(* Logix 5000 project; controller reports 1756-L63 rev 20.11; software revision 20.04; part 50 of 52 *)

        [182].log_data[31].max := 1.0, [182].log_data[31].total := 1629.7471, [182].log_data[31].time := 3600.0, [182].log_data[31].maxminute := 5, [182].log_data[31].valid := 1, [182].log_data[32].max := 1.0, [182].log_data[32].total := 1288.2471, [182].log_data[32].time := 3600.0, [182].log_data[32].maxminute := 2, [182].log_data[32].valid := 1, [182].log_data[33].time := 3600.0, [182].log_data[33].valid := 1, [182].log_data[34].time := 3600.0, [182].log_data[34].valid := 1, [182].log_data[35].max := 1.0, [182].log_data[35].total := 1629.7471, [182].log_data[35].time := 3600.0, [182].log_data[35].maxminute := 8, [182].log_data[35].valid := 1, [182].log_data[36].max := 1.0, [182].log_data[36].total := 1355.247, [182].log_data[36].time := 3600.0, [182].log_data[36].maxminute := 2, [182].log_data[36].valid := 1, [182].log_data[37].max := 7.52496, [182].log_data[37].total := 2850.735, [182].log_data[37].time := 3600.0, [182].log_data[37].minminute := 6, [182].log_data[37].valid := 1, [182].log_data[38].time := 3600.0, [182].log_data[38].valid := 1, [182].log_data[39].min := 0.9950596, [182].log_data[39].max := 1.0219122, [182].log_data[39].total := 3611.1082, [182].log_data[39].time := 3600.0, [182].log_data[39].minminute := 24, [182].log_data[39].maxminute := 6, [182].log_data[39].valid := 1, [182].log_data[40].min := 7.5459046, [182].log_data[40].max := 7.5849276, [182].log_data[40].total := 27253.14, [182].log_data[40].time := 3600.0, [182].log_data[40].minminute := 44, [182].log_data[40].maxminute := 47, [182].log_data[40].valid := 1, [182].log_data[41].min := 0.06945386, [182].log_data[41].max := 0.103412114, [182].log_data[41].total := 295.7068, [182].log_data[41].time := 3600.0, [182].log_data[41].minminute := 41, [182].log_data[41].valid := 1, [182].log_data[42].min := 2.292467, [182].log_data[42].max := 2.2978847, [182].log_data[42].total := 8263.784, [182].log_data[42].time := 3600.0, [182].log_data[42].minminute := 25, [182].log_data[42].valid := 1, [182].log_data[43].min := -0.26000214, [182].log_data[43].max := -0.23999786, [182].log_data[43].total := -935.9582,
        [182].log_data[43].time := 3600.0, [182].log_data[43].maxminute := 40, [182].log_data[43].valid := 1, [182].log_data[44].min := -0.30000305, [182].log_data[44].max := -0.27999878, [182].log_data[44].total := -1034.0974, [182].log_data[44].time := 3600.0, [182].log_data[44].valid := 1, [182].log_data[45].time := 3600.0, [182].log_data[45].valid := 1, [182].log_data[46].time := 3600.0, [182].log_data[46].valid := 1, [182].log_data[47].time := 3600.0, [182].log_data[47].valid := 1, [182].log_data[48].min := 6.578031, [182].log_data[48].max := 6.975128, [182].log_data[48].total := 24224.42, [182].log_data[48].time := 3600.0, [182].log_data[48].minminute := 30, [182].log_data[48].maxminute := 8, [182].log_data[48].valid := 1, [182].log_data[49].min := 6.7680936, [182].log_data[49].max := 9.480644, [182].log_data[49].total := 29086.424, [182].log_data[49].time := 3600.0, [182].log_data[49].minminute := 27, [182].log_data[49].valid := 1, [182].log_data[50].min := 2.0458467, [182].log_data[50].max := 2.1517262, [182].log_data[50].total := 7513.503, [182].log_data[50].time := 3600.0, [182].log_data[50].minminute := 58, [182].log_data[50].maxminute := 2, [182].log_data[50].valid := 1, [182].log_data[51].time := 3600.0, [182].log_data[51].valid := 1, [182].log_data[52].min := -4.199997, [182].log_data[52].max := 0.13999939, [182].log_data[52].total := -7374.407, [182].log_data[52].time := 3600.0, [182].log_data[52].minminute := 2, [182].log_data[52].maxminute := 56, [182].log_data[52].valid := 1, [182].log_data[53].min := -3.9799957, [182].log_data[53].max := 0.27999878, [182].log_data[53].total := -6905.0986, [182].log_data[53].time := 3600.0, [182].log_data[53].minminute := 2, [182].log_data[53].maxminute := 28, [182].log_data[53].valid := 1, [182].log_data[54].max := 0.538, [182].log_data[54].total := 1154.3633, [182].log_data[54].time := 3600.0, [182].log_data[54].maxminute := 16, [182].log_data[54].valid := 1, [182].log_data[55].max := 0.5285, [182].log_data[55].total := 1182.999, [182].log_data[55].time := 3600.0, [182].log_data[55].maxminute := 19, [182].log_data[55].valid := 1,
        [182].log_data[56].min := 0.16044189, [182].log_data[56].max := 0.16087373, [182].log_data[56].total := 578.1737, [182].log_data[56].time := 3600.0, [182].log_data[56].minminute := 7, [182].log_data[56].maxminute := 25, [182].log_data[56].valid := 1, [182].log_data[57].min := 0.34067667, [182].log_data[57].max := 0.34228623, [182].log_data[57].total := 1229.2501, [182].log_data[57].time := 3600.0, [182].log_data[57].minminute := 45, [182].log_data[57].maxminute := 11, [182].log_data[57].valid := 1, [182].log_data[58].time := 3600.0, [182].log_data[58].valid := 1, [182].log_data[59].time := 3600.0, [182].log_data[59].valid := 1, [182].log_data[60].valid := 1, [182].log_data[61].valid := 1, [182].log_data[62].valid := 1, [182].log_data[63].valid := 1, [182].log_data[64].valid := 1, [182].log_data[65].valid := 1, [182].log_data[66].valid := 1, [182].log_data[67].valid := 1, [182].log_data[68].valid := 1, [182].log_data[69].valid := 1, [182].log_data[70].valid := 1, [182].log_data[71].valid := 1, [182].log_data[72].valid := 1, [182].log_data[73].valid := 1, [182].log_data[74].valid := 1, [182].log_data[75].valid := 1, [182].log_data[76].valid := 1, [182].log_data[77].valid := 1, [182].log_data[78].valid := 1, [182].log_data[79].valid := 1, [182].log_data[80].valid := 1, [182].log_data[81].valid := 1, [182].log_data[82].valid := 1, [182].log_data[83].valid := 1, [182].log_data[84].valid := 1, [182].log_data[85].valid := 1, [182].log_data[86].valid := 1, [182].log_data[87].valid := 1, [182].log_data[88].valid := 1, [182].log_data[89].valid := 1, [182].log_data[90].valid := 1, [182].log_data[91].valid := 1, [182].log_data[92].valid := 1, [182].log_data[93].valid := 1, [182].log_data[94].valid := 1, [182].log_data[95].valid := 1, [182].log_data[96].valid := 1, [182].log_data[97].valid := 1, [182].log_data[98].valid := 1, [182].log_data[99].valid := 1, [182].log_data[100].valid := 1, [182].log_data[101].valid := 1,
        [182].log_data[102].valid := 1, [182].log_data[103].valid := 1, [182].log_data[104].valid := 1, [182].log_data[105].valid := 1, [182].log_data[106].valid := 1, [182].log_data[107].valid := 1, [182].log_data[108].valid := 1, [182].log_data[109].valid := 1, [182].log_data[110].valid := 1, [182].log_data[111].valid := 1, [182].log_data[112].valid := 1, [182].log_data[113].valid := 1, [182].log_data[114].valid := 1, [182].log_data[115].valid := 1, [182].log_data[116].valid := 1, [182].log_data[117].valid := 1, [182].log_data[118].valid := 1, [182].log_data[119].valid := 1, [182].log_data[120].valid := 1, [182].log_data[121].valid := 1, [182].log_data[122].valid := 1, [182].log_data[123].valid := 1, [182].log_data[124].valid := 1, [182].time.Year := 2023, [182].time.Month := 1, [182].time.Day := 12, [182].time.Hour := 9, [182].time.Minute := 59, [182].time.Second := 59, [183].log_data[0].min := 1.0, [183].log_data[0].max := 1.0, [183].log_data[0].total := 3600.0, [183].log_data[0].time := 3600.0, [183].log_data[0].valid := 1, [183].log_data[1].max := 1.0, [183].log_data[1].total := 590.5, [183].log_data[1].time := 3600.0, [183].log_data[1].maxminute := 32, [183].log_data[1].valid := 1, [183].log_data[2].max := 1.0, [183].log_data[2].total := 587.0, [183].log_data[2].time := 3600.0, [183].log_data[2].maxminute := 32, [183].log_data[2].valid := 1, [183].log_data[3].time := 3600.0, [183].log_data[3].valid := 1, [183].log_data[4].time := 3600.0, [183].log_data[4].valid := 1, [183].log_data[5].max := 1.0, [183].log_data[5].total := 226.5, [183].log_data[5].time := 3600.0, [183].log_data[5].maxminute := 34, [183].log_data[5].valid := 1, [183].log_data[6].time := 3600.0, [183].log_data[6].valid := 1, [183].log_data[7].time := 3600.0, [183].log_data[7].valid := 1, [183].log_data[8].max := 1.0, [183].log_data[8].total := 3318.0, [183].log_data[8].time := 3600.0,
        [183].log_data[8].minminute := 32, [183].log_data[8].valid := 1, [183].log_data[9].max := 1.0, [183].log_data[9].total := 3314.5, [183].log_data[9].time := 3600.0, [183].log_data[9].minminute := 32, [183].log_data[9].valid := 1, [183].log_data[10].min := 1.0, [183].log_data[10].max := 1.0, [183].log_data[10].total := 3600.0, [183].log_data[10].time := 3600.0, [183].log_data[10].valid := 1, [183].log_data[11].time := 3600.0, [183].log_data[11].valid := 1, [183].log_data[12].min := 1.0, [183].log_data[12].max := 1.0, [183].log_data[12].total := 3600.0, [183].log_data[12].time := 3600.0, [183].log_data[12].valid := 1, [183].log_data[13].min := 1.0, [183].log_data[13].max := 1.0, [183].log_data[13].total := 3600.0, [183].log_data[13].time := 3600.0, [183].log_data[13].valid := 1, [183].log_data[14].time := 3600.0, [183].log_data[14].valid := 1, [183].log_data[15].time := 3600.0, [183].log_data[15].valid := 1, [183].log_data[16].time := 3600.0, [183].log_data[16].valid := 1, [183].log_data[17].min := 1.0, [183].log_data[17].max := 1.0, [183].log_data[17].total := 3600.0, [183].log_data[17].time := 3600.0, [183].log_data[17].valid := 1, [183].log_data[18].time := 3600.0, [183].log_data[18].valid := 1, [183].log_data[19].time := 3600.0, [183].log_data[19].valid := 1, [183].log_data[20].time := 3600.0, [183].log_data[20].valid := 1, [183].log_data[21].min := 1.0, [183].log_data[21].max := 1.0, [183].log_data[21].total := 3600.0, [183].log_data[21].time := 3600.0, [183].log_data[21].valid := 1, [183].log_data[22].time := 3600.0, [183].log_data[22].valid := 1, [183].log_data[23].time := 3600.0, [183].log_data[23].valid := 1, [183].log_data[24].time := 3600.0, [183].log_data[24].valid := 1, [183].log_data[25].time := 3600.0, [183].log_data[25].valid := 1, [183].log_data[26].time := 3600.0, [183].log_data[26].valid := 1, [183].log_data[27].time := 3600.0, [183].log_data[27].valid := 1, [183].log_data[28].time := 3600.0, [183].log_data[28].valid := 1,
        [183].log_data[29].min := 1.0, [183].log_data[29].max := 1.0, [183].log_data[29].total := 3600.0, [183].log_data[29].time := 3600.0, [183].log_data[29].valid := 1, [183].log_data[30].min := 1.0, [183].log_data[30].max := 1.0, [183].log_data[30].total := 3600.0, [183].log_data[30].time := 3600.0, [183].log_data[30].valid := 1, [183].log_data[31].max := 1.0, [183].log_data[31].total := 1268.7471, [183].log_data[31].time := 3600.0, [183].log_data[31].maxminute := 8, [183].log_data[31].valid := 1, [183].log_data[32].max := 1.0, [183].log_data[32].total := 1604.7471, [183].log_data[32].time := 3600.0, [183].log_data[32].minminute := 7, [183].log_data[32].valid := 1, [183].log_data[33].time := 3600.0, [183].log_data[33].valid := 1, [183].log_data[34].time := 3600.0, [183].log_data[34].valid := 1, [183].log_data[35].max := 1.0, [183].log_data[35].total := 1172.2471, [183].log_data[35].time := 3600.0, [183].log_data[35].maxminute := 11, [183].log_data[35].valid := 1, [183].log_data[36].max := 1.0, [183].log_data[36].total := 1629.998, [183].log_data[36].time := 3600.0, [183].log_data[36].maxminute := 1, [183].log_data[36].valid := 1, [183].log_data[37].max := 6.980448, [183].log_data[37].total := 3611.7107, [183].log_data[37].time := 3600.0, [183].log_data[37].maxminute := 33, [183].log_data[37].valid := 1, [183].log_data[38].time := 3600.0, [183].log_data[38].valid := 1, [183].log_data[39].min := 0.9967084, [183].log_data[39].max := 1.0206168, [183].log_data[39].total := 3614.8816, [183].log_data[39].time := 3600.0, [183].log_data[39].minminute := 13, [183].log_data[39].maxminute := 35, [183].log_data[39].valid := 1, [183].log_data[40].min := 7.5316143, [183].log_data[40].max := 7.5849276, [183].log_data[40].total := 27245.064, [183].log_data[40].time := 3600.0, [183].log_data[40].minminute := 25, [183].log_data[40].maxminute := 52, [183].log_data[40].valid := 1, [183].log_data[41].min := 0.0686687, [183].log_data[41].max := 0.09438281, [183].log_data[41].total := 279.35208, [183].log_data[41].time := 3600.0, [183].log_data[41].minminute := 53,
        [183].log_data[41].maxminute := 2, [183].log_data[41].valid := 1, [183].log_data[42].min := 2.2927027, [183].log_data[42].max := 2.297767, [183].log_data[42].total := 8263.784, [183].log_data[42].time := 3600.0, [183].log_data[42].minminute := 5, [183].log_data[42].maxminute := 6, [183].log_data[42].valid := 1, [183].log_data[43].min := -0.26000214, [183].log_data[43].max := -0.23999786, [183].log_data[43].total := -935.8381, [183].log_data[43].time := 3600.0, [183].log_data[43].maxminute := 2, [183].log_data[43].valid := 1, [183].log_data[44].min := -0.30000305, [183].log_data[44].max := -0.27999878, [183].log_data[44].total := -1026.5973, [183].log_data[44].time := 3600.0, [183].log_data[44].valid := 1, [183].log_data[45].time := 3600.0, [183].log_data[45].valid := 1, [183].log_data[46].time := 3600.0, [183].log_data[46].valid := 1, [183].log_data[47].time := 3600.0, [183].log_data[47].valid := 1, [183].log_data[48].min := 6.5824285, [183].log_data[48].max := 6.957815, [183].log_data[48].total := 24226.725, [183].log_data[48].time := 3600.0, [183].log_data[48].minminute := 59, [183].log_data[48].maxminute := 37, [183].log_data[48].valid := 1, [183].log_data[49].min := 6.8424883, [183].log_data[49].max := 9.4459, [183].log_data[49].total := 31391.893, [183].log_data[49].time := 3600.0, [183].log_data[49].minminute := 58, [183].log_data[49].maxminute := 22, [183].log_data[49].valid := 1, [183].log_data[50].min := 1.9999144, [183].log_data[50].max := 2.1501951, [183].log_data[50].total := 7404.694, [183].log_data[50].time := 3600.0, [183].log_data[50].minminute := 32, [183].log_data[50].maxminute := 37, [183].log_data[50].valid := 1, [183].log_data[51].time := 3600.0, [183].log_data[51].valid := 1, [183].log_data[52].min := -3.8600006, [183].log_data[52].max := 0.13999939, [183].log_data[52].total := -7261.7637, [183].log_data[52].time := 3600.0, [183].log_data[52].minminute := 37, [183].log_data[52].maxminute := 7, [183].log_data[52].valid := 1, [183].log_data[53].min := -3.7200012, [183].log_data[53].max := 0.22000122, [183].log_data[53].total := -6467.2256, [183].log_data[53].time := 3600.0,
        [183].log_data[53].minminute := 37, [183].log_data[53].valid := 1, [183].log_data[54].max := 0.52349997, [183].log_data[54].total := 1138.3706, [183].log_data[54].time := 3600.0, [183].log_data[54].minminute := 7, [183].log_data[54].maxminute := 55, [183].log_data[54].valid := 1, [183].log_data[55].max := 0.5395, [183].log_data[55].total := 1109.6932, [183].log_data[55].time := 3600.0, [183].log_data[55].maxminute := 11, [183].log_data[55].valid := 1, [183].log_data[56].min := 0.16044189, [183].log_data[56].max := 0.16083448, [183].log_data[56].total := 578.1302, [183].log_data[56].time := 3600.0, [183].log_data[56].minminute := 22, [183].log_data[56].maxminute := 1, [183].log_data[56].valid := 1, [183].log_data[57].min := 0.34040186, [183].log_data[57].max := 0.34106925, [183].log_data[57].total := 1226.9022, [183].log_data[57].time := 3600.0, [183].log_data[57].minminute := 59, [183].log_data[57].maxminute := 18, [183].log_data[57].valid := 1, [183].log_data[58].time := 3600.0, [183].log_data[58].valid := 1, [183].log_data[59].time := 3600.0, [183].log_data[59].valid := 1, [183].log_data[60].valid := 1, [183].log_data[61].valid := 1, [183].log_data[62].valid := 1, [183].log_data[63].valid := 1, [183].log_data[64].valid := 1, [183].log_data[65].valid := 1, [183].log_data[66].valid := 1, [183].log_data[67].valid := 1, [183].log_data[68].valid := 1, [183].log_data[69].valid := 1, [183].log_data[70].valid := 1, [183].log_data[71].valid := 1, [183].log_data[72].valid := 1, [183].log_data[73].valid := 1, [183].log_data[74].valid := 1, [183].log_data[75].valid := 1, [183].log_data[76].valid := 1, [183].log_data[77].valid := 1, [183].log_data[78].valid := 1, [183].log_data[79].valid := 1, [183].log_data[80].valid := 1, [183].log_data[81].valid := 1, [183].log_data[82].valid := 1, [183].log_data[83].valid := 1, [183].log_data[84].valid := 1, [183].log_data[85].valid := 1, [183].log_data[86].valid := 1, [183].log_data[87].valid := 1, [183].log_data[88].valid := 1,
        [183].log_data[89].valid := 1, [183].log_data[90].valid := 1, [183].log_data[91].valid := 1, [183].log_data[92].valid := 1, [183].log_data[93].valid := 1, [183].log_data[94].valid := 1, [183].log_data[95].valid := 1, [183].log_data[96].valid := 1, [183].log_data[97].valid := 1, [183].log_data[98].valid := 1, [183].log_data[99].valid := 1, [183].log_data[100].valid := 1, [183].log_data[101].valid := 1, [183].log_data[102].valid := 1, [183].log_data[103].valid := 1, [183].log_data[104].valid := 1, [183].log_data[105].valid := 1, [183].log_data[106].valid := 1, [183].log_data[107].valid := 1, [183].log_data[108].valid := 1, [183].log_data[109].valid := 1, [183].log_data[110].valid := 1, [183].log_data[111].valid := 1, [183].log_data[112].valid := 1, [183].log_data[113].valid := 1, [183].log_data[114].valid := 1, [183].log_data[115].valid := 1, [183].log_data[116].valid := 1, [183].log_data[117].valid := 1, [183].log_data[118].valid := 1, [183].log_data[119].valid := 1, [183].log_data[120].valid := 1, [183].log_data[121].valid := 1, [183].log_data[122].valid := 1, [183].log_data[123].valid := 1, [183].log_data[124].valid := 1, [183].time.Year := 2023, [183].time.Month := 1, [183].time.Day := 12, [183].time.Hour := 10, [183].time.Minute := 59, [183].time.Second := 59, [184].log_data[0].min := 1.0, [184].log_data[0].max := 1.0, [184].log_data[0].total := 3600.0, [184].log_data[0].time := 3600.0, [184].log_data[0].valid := 1, [184].log_data[1].time := 3600.0, [184].log_data[1].valid := 1, [184].log_data[2].time := 3600.0, [184].log_data[2].valid := 1, [184].log_data[3].time := 3600.0, [184].log_data[3].valid := 1, [184].log_data[4].time := 3600.0, [184].log_data[4].valid := 1, [184].log_data[5].time := 3600.0, [184].log_data[5].valid := 1, [184].log_data[6].time := 3600.0, [184].log_data[6].valid := 1, [184].log_data[7].time := 3600.0,
        [184].log_data[7].valid := 1, [184].log_data[8].min := 1.0, [184].log_data[8].max := 1.0, [184].log_data[8].total := 3600.0, [184].log_data[8].time := 3600.0, [184].log_data[8].valid := 1, [184].log_data[9].min := 1.0, [184].log_data[9].max := 1.0, [184].log_data[9].total := 3600.0, [184].log_data[9].time := 3600.0, [184].log_data[9].valid := 1, [184].log_data[10].min := 1.0, [184].log_data[10].max := 1.0, [184].log_data[10].total := 3600.0, [184].log_data[10].time := 3600.0, [184].log_data[10].valid := 1, [184].log_data[11].time := 3600.0, [184].log_data[11].valid := 1, [184].log_data[12].min := 1.0, [184].log_data[12].max := 1.0, [184].log_data[12].total := 3600.0, [184].log_data[12].time := 3600.0, [184].log_data[12].valid := 1, [184].log_data[13].min := 1.0, [184].log_data[13].max := 1.0, [184].log_data[13].total := 3600.0, [184].log_data[13].time := 3600.0, [184].log_data[13].valid := 1, [184].log_data[14].time := 3600.0, [184].log_data[14].valid := 1, [184].log_data[15].time := 3600.0, [184].log_data[15].valid := 1, [184].log_data[16].time := 3600.0, [184].log_data[16].valid := 1, [184].log_data[17].min := 1.0, [184].log_data[17].max := 1.0, [184].log_data[17].total := 3600.0, [184].log_data[17].time := 3600.0, [184].log_data[17].valid := 1, [184].log_data[18].time := 3600.0, [184].log_data[18].valid := 1, [184].log_data[19].time := 3600.0, [184].log_data[19].valid := 1, [184].log_data[20].time := 3600.0, [184].log_data[20].valid := 1, [184].log_data[21].min := 1.0, [184].log_data[21].max := 1.0, [184].log_data[21].total := 3600.0, [184].log_data[21].time := 3600.0, [184].log_data[21].valid := 1, [184].log_data[22].time := 3600.0, [184].log_data[22].valid := 1, [184].log_data[23].time := 3600.0, [184].log_data[23].valid := 1, [184].log_data[24].time := 3600.0, [184].log_data[24].valid := 1, [184].log_data[25].time := 3600.0, [184].log_data[25].valid := 1, [184].log_data[26].time := 3600.0, [184].log_data[26].valid := 1,
        [184].log_data[27].time := 3600.0, [184].log_data[27].valid := 1, [184].log_data[28].time := 3600.0, [184].log_data[28].valid := 1, [184].log_data[29].min := 1.0, [184].log_data[29].max := 1.0, [184].log_data[29].total := 3600.0, [184].log_data[29].time := 3600.0, [184].log_data[29].valid := 1, [184].log_data[30].min := 1.0, [184].log_data[30].max := 1.0, [184].log_data[30].total := 3600.0, [184].log_data[30].time := 3600.0, [184].log_data[30].valid := 1, [184].log_data[31].max := 1.0, [184].log_data[31].total := 1629.998, [184].log_data[31].time := 3600.0, [184].log_data[31].maxminute := 5, [184].log_data[31].valid := 1, [184].log_data[32].max := 1.0, [184].log_data[32].total := 1440.498, [184].log_data[32].time := 3600.0, [184].log_data[32].minminute := 4, [184].log_data[32].valid := 1, [184].log_data[33].time := 3600.0, [184].log_data[33].valid := 1, [184].log_data[34].time := 3600.0, [184].log_data[34].valid := 1, [184].log_data[35].max := 1.0, [184].log_data[35].total := 1543.998, [184].log_data[35].time := 3600.0, [184].log_data[35].minminute := 7, [184].log_data[35].valid := 1, [184].log_data[36].max := 1.0, [184].log_data[36].total := 1614.7471, [184].log_data[36].time := 3600.0, [184].log_data[36].maxminute := 9, [184].log_data[36].valid := 1, [184].log_data[37].time := 3600.0, [184].log_data[37].valid := 1, [184].log_data[38].time := 3600.0, [184].log_data[38].valid := 1, [184].log_data[39].min := 1.000595, [184].log_data[39].max := 1.0097814, [184].log_data[39].total := 3621.283, [184].log_data[39].time := 3600.0, [184].log_data[39].minminute := 56, [184].log_data[39].maxminute := 32, [184].log_data[39].valid := 1, [184].log_data[40].min := 7.530241, [184].log_data[40].max := 7.590423, [184].log_data[40].total := 27254.365, [184].log_data[40].time := 3600.0, [184].log_data[40].minminute := 14, [184].log_data[40].maxminute := 2, [184].log_data[40].valid := 1, [184].log_data[41].min := 0.071613036, [184].log_data[41].max := 0.10674902, [184].log_data[41].total := 300.04837, [184].log_data[41].time := 3600.0,
        [184].log_data[41].minminute := 57, [184].log_data[41].maxminute := 12, [184].log_data[41].valid := 1, [184].log_data[42].min := 2.2928205, [184].log_data[42].max := 2.2978847, [184].log_data[42].total := 8263.812, [184].log_data[42].time := 3600.0, [184].log_data[42].minminute := 40, [184].log_data[42].maxminute := 35, [184].log_data[42].valid := 1, [184].log_data[43].min := -0.26000214, [184].log_data[43].max := -0.23999786, [184].log_data[43].total := -935.8931, [184].log_data[43].time := 3600.0, [184].log_data[43].maxminute := 5, [184].log_data[43].valid := 1, [184].log_data[44].min := -0.30000305, [184].log_data[44].max := -0.27999878, [184].log_data[44].total := -1037.5183, [184].log_data[44].time := 3600.0, [184].log_data[44].valid := 1, [184].log_data[45].time := 3600.0, [184].log_data[45].valid := 1, [184].log_data[46].time := 3600.0, [184].log_data[46].valid := 1, [184].log_data[47].time := 3600.0, [184].log_data[47].valid := 1, [184].log_data[48].min := 6.5766573, [184].log_data[48].max := 6.788259, [184].log_data[48].total := 24232.771, [184].log_data[48].time := 3600.0, [184].log_data[48].minminute := 2, [184].log_data[48].maxminute := 16, [184].log_data[48].valid := 1, [184].log_data[49].min := 6.8424883, [184].log_data[49].max := 9.414298, [184].log_data[49].total := 31253.555, [184].log_data[49].time := 3600.0, [184].log_data[49].maxminute := 54, [184].log_data[49].valid := 1, [184].log_data[50].min := 2.0008566, [184].log_data[50].max := 2.0907187, [184].log_data[50].total := 7364.591, [184].log_data[50].time := 3600.0, [184].log_data[50].minminute := 59, [184].log_data[50].valid := 1, [184].log_data[51].time := 3600.0, [184].log_data[51].valid := 1, [184].log_data[52].min := -2.8600006, [184].log_data[52].max := 0.13999939, [184].log_data[52].total := -7446.0986, [184].log_data[52].time := 3600.0, [184].log_data[52].minminute := 6, [184].log_data[52].maxminute := 4, [184].log_data[52].valid := 1, [184].log_data[53].min := -2.4800034, [184].log_data[53].max := 0.2599945, [184].log_data[53].total := -7103.2104, [184].log_data[53].time := 3600.0, [184].log_data[53].minminute := 21,
        [184].log_data[53].maxminute := 50, [184].log_data[53].valid := 1, [184].log_data[54].max := 0.5525, [184].log_data[54].total := 1217.0905, [184].log_data[54].time := 3600.0, [184].log_data[54].minminute := 4, [184].log_data[54].maxminute := 6, [184].log_data[54].valid := 1, [184].log_data[55].max := 0.5205, [184].log_data[55].total := 1254.2858, [184].log_data[55].time := 3600.0, [184].log_data[55].minminute := 7, [184].log_data[55].maxminute := 19, [184].log_data[55].valid := 1, [184].log_data[56].min := 0.16040264, [184].log_data[56].max := 0.16079521, [184].log_data[56].total := 578.0307, [184].log_data[56].time := 3600.0, [184].log_data[56].minminute := 26, [184].log_data[56].maxminute := 4, [184].log_data[56].valid := 1, [184].log_data[57].min := 0.33875299, [184].log_data[57].max := 0.3405589, [184].log_data[57].total := 1220.648, [184].log_data[57].time := 3600.0, [184].log_data[57].minminute := 37, [184].log_data[57].valid := 1, [184].log_data[58].time := 3600.0, [184].log_data[58].valid := 1, [184].log_data[59].time := 3600.0, [184].log_data[59].valid := 1, [184].log_data[60].valid := 1, [184].log_data[61].valid := 1, [184].log_data[62].valid := 1, [184].log_data[63].valid := 1, [184].log_data[64].valid := 1, [184].log_data[65].valid := 1, [184].log_data[66].valid := 1, [184].log_data[67].valid := 1, [184].log_data[68].valid := 1, [184].log_data[69].valid := 1, [184].log_data[70].valid := 1, [184].log_data[71].valid := 1, [184].log_data[72].valid := 1, [184].log_data[73].valid := 1, [184].log_data[74].valid := 1, [184].log_data[75].valid := 1, [184].log_data[76].valid := 1, [184].log_data[77].valid := 1, [184].log_data[78].valid := 1, [184].log_data[79].valid := 1, [184].log_data[80].valid := 1, [184].log_data[81].valid := 1, [184].log_data[82].valid := 1, [184].log_data[83].valid := 1, [184].log_data[84].valid := 1, [184].log_data[85].valid := 1, [184].log_data[86].valid := 1, [184].log_data[87].valid := 1, [184].log_data[88].valid := 1,
        [184].log_data[89].valid := 1, [184].log_data[90].valid := 1, [184].log_data[91].valid := 1, [184].log_data[92].valid := 1, [184].log_data[93].valid := 1, [184].log_data[94].valid := 1, [184].log_data[95].valid := 1, [184].log_data[96].valid := 1, [184].log_data[97].valid := 1, [184].log_data[98].valid := 1, [184].log_data[99].valid := 1, [184].log_data[100].valid := 1, [184].log_data[101].valid := 1, [184].log_data[102].valid := 1, [184].log_data[103].valid := 1, [184].log_data[104].valid := 1, [184].log_data[105].valid := 1, [184].log_data[106].valid := 1, [184].log_data[107].valid := 1, [184].log_data[108].valid := 1, [184].log_data[109].valid := 1, [184].log_data[110].valid := 1, [184].log_data[111].valid := 1, [184].log_data[112].valid := 1, [184].log_data[113].valid := 1, [184].log_data[114].valid := 1, [184].log_data[115].valid := 1, [184].log_data[116].valid := 1, [184].log_data[117].valid := 1, [184].log_data[118].valid := 1, [184].log_data[119].valid := 1, [184].log_data[120].valid := 1, [184].log_data[121].valid := 1, [184].log_data[122].valid := 1, [184].log_data[123].valid := 1, [184].log_data[124].valid := 1, [184].time.Year := 2023, [184].time.Month := 1, [184].time.Day := 12, [184].time.Hour := 11, [184].time.Minute := 59, [184].time.Second := 59, [185].log_data[0].min := 1.0, [185].log_data[0].max := 1.0, [185].log_data[0].total := 3600.0, [185].log_data[0].time := 3600.0, [185].log_data[0].valid := 1, [185].log_data[1].max := 1.0, [185].log_data[1].total := 552.5, [185].log_data[1].time := 3600.0, [185].log_data[1].maxminute := 5, [185].log_data[1].valid := 1, [185].log_data[2].max := 1.0, [185].log_data[2].total := 549.0, [185].log_data[2].time := 3600.0, [185].log_data[2].maxminute := 5, [185].log_data[2].valid := 1, [185].log_data[3].time := 3600.0, [185].log_data[3].valid := 1, [185].log_data[4].time := 3600.0,
        [185].log_data[4].valid := 1, [185].log_data[5].max := 1.0, [185].log_data[5].total := 252.0, [185].log_data[5].time := 3600.0, [185].log_data[5].maxminute := 7, [185].log_data[5].valid := 1, [185].log_data[6].time := 3600.0, [185].log_data[6].valid := 1, [185].log_data[7].time := 3600.0, [185].log_data[7].valid := 1, [185].log_data[8].max := 1.0, [185].log_data[8].total := 3070.5, [185].log_data[8].time := 3600.0, [185].log_data[8].valid := 1, [185].log_data[9].max := 1.0, [185].log_data[9].total := 3067.0, [185].log_data[9].time := 3600.0, [185].log_data[9].valid := 1, [185].log_data[10].min := 1.0, [185].log_data[10].max := 1.0, [185].log_data[10].total := 3600.0, [185].log_data[10].time := 3600.0, [185].log_data[10].valid := 1, [185].log_data[11].time := 3600.0, [185].log_data[11].valid := 1, [185].log_data[12].min := 1.0, [185].log_data[12].max := 1.0, [185].log_data[12].total := 3600.0, [185].log_data[12].time := 3600.0, [185].log_data[12].valid := 1, [185].log_data[13].min := 1.0, [185].log_data[13].max := 1.0, [185].log_data[13].total := 3600.0, [185].log_data[13].time := 3600.0, [185].log_data[13].valid := 1, [185].log_data[14].time := 3600.0, [185].log_data[14].valid := 1, [185].log_data[15].time := 3600.0, [185].log_data[15].valid := 1, [185].log_data[16].time := 3600.0, [185].log_data[16].valid := 1, [185].log_data[17].min := 1.0, [185].log_data[17].max := 1.0, [185].log_data[17].total := 3600.0, [185].log_data[17].time := 3600.0, [185].log_data[17].valid := 1, [185].log_data[18].time := 3600.0, [185].log_data[18].valid := 1, [185].log_data[19].time := 3600.0, [185].log_data[19].valid := 1, [185].log_data[20].time := 3600.0, [185].log_data[20].valid := 1, [185].log_data[21].min := 1.0, [185].log_data[21].max := 1.0, [185].log_data[21].total := 3600.0, [185].log_data[21].time := 3600.0, [185].log_data[21].valid := 1, [185].log_data[22].time := 3600.0, [185].log_data[22].valid := 1, [185].log_data[23].time := 3600.0,
        [185].log_data[23].valid := 1, [185].log_data[24].time := 3600.0, [185].log_data[24].valid := 1, [185].log_data[25].time := 3600.0, [185].log_data[25].valid := 1, [185].log_data[26].time := 3600.0, [185].log_data[26].valid := 1, [185].log_data[27].time := 3600.0, [185].log_data[27].valid := 1, [185].log_data[28].time := 3600.0, [185].log_data[28].valid := 1, [185].log_data[29].min := 1.0, [185].log_data[29].max := 1.0, [185].log_data[29].total := 3600.0, [185].log_data[29].time := 3600.0, [185].log_data[29].valid := 1, [185].log_data[30].min := 1.0, [185].log_data[30].max := 1.0, [185].log_data[30].total := 3600.0, [185].log_data[30].time := 3600.0, [185].log_data[30].valid := 1, [185].log_data[31].max := 1.0, [185].log_data[31].total := 1522.247, [185].log_data[31].time := 3600.0, [185].log_data[31].maxminute := 9, [185].log_data[31].valid := 1, [185].log_data[32].max := 1.0, [185].log_data[32].total := 1112.0, [185].log_data[32].time := 3600.0, [185].log_data[32].valid := 1, [185].log_data[33].time := 3600.0, [185].log_data[33].valid := 1, [185].log_data[34].time := 3600.0, [185].log_data[34].valid := 1, [185].log_data[35].max := 1.0, [185].log_data[35].total := 1598.498, [185].log_data[35].time := 3600.0, [185].log_data[35].maxminute := 9, [185].log_data[35].valid := 1, [185].log_data[36].max := 1.0, [185].log_data[36].total := 1102.0, [185].log_data[36].time := 3600.0, [185].log_data[36].valid := 1, [185].log_data[37].max := 7.5520477, [185].log_data[37].total := 3618.2432, [185].log_data[37].time := 3600.0, [185].log_data[37].maxminute := 6, [185].log_data[37].valid := 1, [185].log_data[38].time := 3600.0, [185].log_data[38].valid := 1, [185].log_data[39].min := 0.99694395, [185].log_data[39].max := 1.0217944, [185].log_data[39].total := 3616.0115, [185].log_data[39].time := 3600.0, [185].log_data[39].minminute := 58, [185].log_data[39].maxminute := 11, [185].log_data[39].valid := 1, [185].log_data[40].min := 7.5373855, [185].log_data[40].max := 7.590698, [185].log_data[40].total := 27249.404,
        [185].log_data[40].time := 3600.0, [185].log_data[40].minminute := 26, [185].log_data[40].maxminute := 12, [185].log_data[40].valid := 1, [185].log_data[41].min := 0.058461428, [185].log_data[41].max := 0.09948633, [185].log_data[41].total := 278.58185, [185].log_data[41].time := 3600.0, [185].log_data[41].minminute := 55, [185].log_data[41].maxminute := 19, [185].log_data[41].valid := 1, [185].log_data[42].min := 2.2929382, [185].log_data[42].max := 2.297767, [185].log_data[42].total := 8263.846, [185].log_data[42].time := 3600.0, [185].log_data[42].minminute := 51, [185].log_data[42].maxminute := 19, [185].log_data[42].valid := 1, [185].log_data[43].min := -0.26000214, [185].log_data[43].max := -0.23999786, [185].log_data[43].total := -935.95825, [185].log_data[43].time := 3600.0, [185].log_data[43].maxminute := 18, [185].log_data[43].valid := 1, [185].log_data[44].min := -0.30000305, [185].log_data[44].max := -0.27999878, [185].log_data[44].total := -1048.6907, [185].log_data[44].time := 3600.0, [185].log_data[44].valid := 1, [185].log_data[45].time := 3600.0, [185].log_data[45].valid := 1, [185].log_data[46].time := 3600.0, [185].log_data[46].valid := 1, [185].log_data[47].time := 3600.0, [185].log_data[47].valid := 1, [185].log_data[48].min := 6.5722604, [185].log_data[48].max := 6.9732046, [185].log_data[48].total := 24212.016, [185].log_data[48].time := 3600.0, [185].log_data[48].minminute := 36, [185].log_data[48].maxminute := 14, [185].log_data[48].valid := 1, [185].log_data[49].min := 6.660133, [185].log_data[49].max := 9.409195, [185].log_data[49].total := 28331.281, [185].log_data[49].time := 3600.0, [185].log_data[49].minminute := 35, [185].log_data[49].maxminute := 6, [185].log_data[49].valid := 1, [185].log_data[50].min := 1.9985011, [185].log_data[50].max := 2.1512551, [185].log_data[50].total := 7526.405, [185].log_data[50].time := 3600.0, [185].log_data[50].maxminute := 9, [185].log_data[50].valid := 1, [185].log_data[51].time := 3600.0, [185].log_data[51].valid := 1, [185].log_data[52].min := -4.040001, [185].log_data[52].max := 0.11999512, [185].log_data[52].total := -7068.036,
        [185].log_data[52].time := 3600.0, [185].log_data[52].minminute := 9, [185].log_data[52].maxminute := 16, [185].log_data[52].valid := 1, [185].log_data[53].min := -3.9799957, [185].log_data[53].max := 0.22000122, [185].log_data[53].total := -6659.7754, [185].log_data[53].time := 3600.0, [185].log_data[53].minminute := 9, [185].log_data[53].maxminute := 19, [185].log_data[53].valid := 1, [185].log_data[54].max := 0.531, [185].log_data[54].total := 1045.1531, [185].log_data[54].time := 3600.0, [185].log_data[54].maxminute := 28, [185].log_data[54].valid := 1, [185].log_data[55].max := 0.559, [185].log_data[55].total := 1071.3711, [185].log_data[55].time := 3600.0, [185].log_data[55].maxminute := 51, [185].log_data[55].valid := 1, [185].log_data[56].min := 0.16036338, [185].log_data[56].max := 0.16075596, [185].log_data[56].total := 577.9964, [185].log_data[56].time := 3600.0, [185].log_data[56].minminute := 38, [185].log_data[56].valid := 1, [185].log_data[57].min := 0.33655453, [185].log_data[57].max := 0.33918485, [185].log_data[57].total := 1217.2412, [185].log_data[57].time := 3600.0, [185].log_data[57].minminute := 51, [185].log_data[57].maxminute := 21, [185].log_data[57].valid := 1, [185].log_data[58].time := 3600.0, [185].log_data[58].valid := 1, [185].log_data[59].time := 3600.0, [185].log_data[59].valid := 1, [185].log_data[60].valid := 1, [185].log_data[61].valid := 1, [185].log_data[62].valid := 1, [185].log_data[63].valid := 1, [185].log_data[64].valid := 1, [185].log_data[65].valid := 1, [185].log_data[66].valid := 1, [185].log_data[67].valid := 1, [185].log_data[68].valid := 1, [185].log_data[69].valid := 1, [185].log_data[70].valid := 1, [185].log_data[71].valid := 1, [185].log_data[72].valid := 1, [185].log_data[73].valid := 1, [185].log_data[74].valid := 1, [185].log_data[75].valid := 1, [185].log_data[76].valid := 1, [185].log_data[77].valid := 1, [185].log_data[78].valid := 1, [185].log_data[79].valid := 1, [185].log_data[80].valid := 1, [185].log_data[81].valid := 1,
        [185].log_data[82].valid := 1, [185].log_data[83].valid := 1, [185].log_data[84].valid := 1, [185].log_data[85].valid := 1, [185].log_data[86].valid := 1, [185].log_data[87].valid := 1, [185].log_data[88].valid := 1, [185].log_data[89].valid := 1, [185].log_data[90].valid := 1, [185].log_data[91].valid := 1, [185].log_data[92].valid := 1, [185].log_data[93].valid := 1, [185].log_data[94].valid := 1, [185].log_data[95].valid := 1, [185].log_data[96].valid := 1, [185].log_data[97].valid := 1, [185].log_data[98].valid := 1, [185].log_data[99].valid := 1, [185].log_data[100].valid := 1, [185].log_data[101].valid := 1, [185].log_data[102].valid := 1, [185].log_data[103].valid := 1, [185].log_data[104].valid := 1, [185].log_data[105].valid := 1, [185].log_data[106].valid := 1, [185].log_data[107].valid := 1, [185].log_data[108].valid := 1, [185].log_data[109].valid := 1, [185].log_data[110].valid := 1, [185].log_data[111].valid := 1, [185].log_data[112].valid := 1, [185].log_data[113].valid := 1, [185].log_data[114].valid := 1, [185].log_data[115].valid := 1, [185].log_data[116].valid := 1, [185].log_data[117].valid := 1, [185].log_data[118].valid := 1, [185].log_data[119].valid := 1, [185].log_data[120].valid := 1, [185].log_data[121].valid := 1, [185].log_data[122].valid := 1, [185].log_data[123].valid := 1, [185].log_data[124].valid := 1, [185].time.Year := 2023, [185].time.Month := 1, [185].time.Day := 12, [185].time.Hour := 12, [185].time.Minute := 59, [185].time.Second := 59, [186].log_data[0].min := 1.0, [186].log_data[0].max := 1.0, [186].log_data[0].total := 3599.5, [186].log_data[0].time := 3599.5, [186].log_data[0].valid := 1, [186].log_data[1].max := 1.0, [186].log_data[1].total := 344.749, [186].log_data[1].time := 3599.5, [186].log_data[1].maxminute := 54, [186].log_data[1].valid := 1, [186].log_data[2].max := 1.0,
        [186].log_data[2].total := 341.249, [186].log_data[2].time := 3599.5, [186].log_data[2].maxminute := 54, [186].log_data[2].valid := 1, [186].log_data[3].time := 3599.5, [186].log_data[3].valid := 1, [186].log_data[4].time := 3599.5, [186].log_data[4].valid := 1, [186].log_data[5].max := 1.0, [186].log_data[5].total := 122.5, [186].log_data[5].time := 3599.5, [186].log_data[5].maxminute := 56, [186].log_data[5].valid := 1, [186].log_data[6].time := 3599.5, [186].log_data[6].valid := 1, [186].log_data[7].time := 3599.5, [186].log_data[7].valid := 1, [186].log_data[8].max := 1.0, [186].log_data[8].total := 2593.0, [186].log_data[8].time := 3599.5, [186].log_data[8].minminute := 41, [186].log_data[8].valid := 1, [186].log_data[9].max := 1.0, [186].log_data[9].total := 2589.5, [186].log_data[9].time := 3599.5, [186].log_data[9].minminute := 41, [186].log_data[9].valid := 1, [186].log_data[10].min := 1.0, [186].log_data[10].max := 1.0, [186].log_data[10].total := 3599.5, [186].log_data[10].time := 3599.5, [186].log_data[10].valid := 1, [186].log_data[11].time := 3599.5, [186].log_data[11].valid := 1, [186].log_data[12].min := 1.0, [186].log_data[12].max := 1.0, [186].log_data[12].total := 3599.5, [186].log_data[12].time := 3599.5, [186].log_data[12].valid := 1, [186].log_data[13].min := 1.0, [186].log_data[13].max := 1.0, [186].log_data[13].total := 3599.5, [186].log_data[13].time := 3599.5, [186].log_data[13].valid := 1, [186].log_data[14].time := 3599.5, [186].log_data[14].valid := 1, [186].log_data[15].time := 3599.5, [186].log_data[15].valid := 1, [186].log_data[16].time := 3599.5, [186].log_data[16].valid := 1, [186].log_data[17].min := 1.0, [186].log_data[17].max := 1.0, [186].log_data[17].total := 3599.5, [186].log_data[17].time := 3599.5, [186].log_data[17].valid := 1, [186].log_data[18].time := 3599.5, [186].log_data[18].valid := 1, [186].log_data[19].time := 3599.5, [186].log_data[19].valid := 1, [186].log_data[20].time := 3599.5,
        [186].log_data[20].valid := 1, [186].log_data[21].min := 1.0, [186].log_data[21].max := 1.0, [186].log_data[21].total := 3599.5, [186].log_data[21].time := 3599.5, [186].log_data[21].valid := 1, [186].log_data[22].time := 3599.5, [186].log_data[22].valid := 1, [186].log_data[23].time := 3599.5, [186].log_data[23].valid := 1, [186].log_data[24].time := 3599.5, [186].log_data[24].valid := 1, [186].log_data[25].time := 3599.5, [186].log_data[25].valid := 1, [186].log_data[26].time := 3599.5, [186].log_data[26].valid := 1, [186].log_data[27].time := 3599.5, [186].log_data[27].valid := 1, [186].log_data[28].time := 3599.5, [186].log_data[28].valid := 1, [186].log_data[29].min := 1.0, [186].log_data[29].max := 1.0, [186].log_data[29].total := 3599.5, [186].log_data[29].time := 3599.5, [186].log_data[29].valid := 1, [186].log_data[30].min := 1.0, [186].log_data[30].max := 1.0, [186].log_data[30].total := 3599.5, [186].log_data[30].time := 3599.5, [186].log_data[30].valid := 1, [186].log_data[31].max := 1.0, [186].log_data[31].total := 1086.498, [186].log_data[31].time := 3599.5, [186].log_data[31].maxminute := 10, [186].log_data[31].valid := 1, [186].log_data[32].max := 1.0, [186].log_data[32].total := 1186.2471, [186].log_data[32].time := 3599.5, [186].log_data[32].valid := 1, [186].log_data[33].time := 3599.5, [186].log_data[33].valid := 1, [186].log_data[34].time := 3599.5, [186].log_data[34].valid := 1, [186].log_data[35].max := 1.0, [186].log_data[35].total := 1050.498, [186].log_data[35].time := 3599.5, [186].log_data[35].valid := 1, [186].log_data[36].max := 1.0, [186].log_data[36].total := 1153.7471, [186].log_data[36].time := 3599.5, [186].log_data[36].maxminute := 2, [186].log_data[36].valid := 1, [186].log_data[37].max := 6.989477, [186].log_data[37].total := 2357.3582, [186].log_data[37].time := 3599.5, [186].log_data[37].maxminute := 55, [186].log_data[37].valid := 1, [186].log_data[38].time := 3599.5, [186].log_data[38].valid := 1, [186].log_data[39].min := 0.99753284,
        [186].log_data[39].max := 1.0212055, [186].log_data[39].total := 3613.32, [186].log_data[39].time := 3599.5, [186].log_data[39].minminute := 36, [186].log_data[39].maxminute := 56, [186].log_data[39].valid := 1, [186].log_data[40].min := 7.5459046, [186].log_data[40].max := 7.5934467, [186].log_data[40].total := 27253.635, [186].log_data[40].time := 3599.5, [186].log_data[40].maxminute := 5, [186].log_data[40].valid := 1, [186].log_data[41].min := 0.056498535, [186].log_data[41].max := 0.08829786, [186].log_data[41].total := 249.71246, [186].log_data[41].time := 3599.5, [186].log_data[41].minminute := 20, [186].log_data[41].maxminute := 23, [186].log_data[41].valid := 1, [186].log_data[42].min := 2.292467, [186].log_data[42].max := 2.297767, [186].log_data[42].total := 8262.826, [186].log_data[42].time := 3599.5, [186].log_data[42].minminute := 39, [186].log_data[42].maxminute := 44, [186].log_data[42].valid := 1, [186].log_data[43].min := -0.26000214, [186].log_data[43].max := -0.26000214, [186].log_data[43].total := -935.8432, [186].log_data[43].time := 3599.5, [186].log_data[43].valid := 1, [186].log_data[44].min := -0.30000305, [186].log_data[44].max := -0.27999878, [186].log_data[44].total := -1052.3257, [186].log_data[44].time := 3599.5, [186].log_data[44].valid := 1, [186].log_data[45].time := 3599.5, [186].log_data[45].valid := 1, [186].log_data[46].time := 3599.5, [186].log_data[46].valid := 1, [186].log_data[47].time := 3599.5, [186].log_data[47].valid := 1, [186].log_data[48].min := 6.743465, [186].log_data[48].max := 6.903678, [186].log_data[48].total := 24325.06, [186].log_data[48].time := 3599.5, [186].log_data[48].minminute := 44, [186].log_data[48].maxminute := 59, [186].log_data[48].valid := 1, [186].log_data[49].min := 8.798139, [186].log_data[49].max := 9.401342, [186].log_data[49].total := 33422.215, [186].log_data[49].time := 3599.5, [186].log_data[49].minminute := 59, [186].log_data[49].maxminute := 32, [186].log_data[49].valid := 1, [186].log_data[50].min := 1.9987367, [186].log_data[50].max := 2.1501951, [186].log_data[50].total := 7385.422, [186].log_data[50].time := 3599.5,
        [186].log_data[50].minminute := 41, [186].log_data[50].maxminute := 58, [186].log_data[50].valid := 1, [186].log_data[51].time := 3599.5, [186].log_data[51].valid := 1, [186].log_data[52].min := -4.119995, [186].log_data[52].max := 0.13999939, [186].log_data[52].total := -6856.9106, [186].log_data[52].time := 3599.5, [186].log_data[52].minminute := 58, [186].log_data[52].maxminute := 9, [186].log_data[52].valid := 1, [186].log_data[53].min := -3.899994, [186].log_data[53].max := 0.22000122, [186].log_data[53].total := -6188.398, [186].log_data[53].time := 3599.5, [186].log_data[53].minminute := 58, [186].log_data[53].maxminute := 2, [186].log_data[53].valid := 1, [186].log_data[54].max := 0.518, [186].log_data[54].total := 899.5263, [186].log_data[54].time := 3599.5, [186].log_data[54].maxminute := 10, [186].log_data[54].valid := 1, [186].log_data[55].max := 0.5335, [186].log_data[55].total := 872.8351, [186].log_data[55].time := 3599.5, [186].log_data[55].maxminute := 12, [186].log_data[55].valid := 1, [186].log_data[56].min := 0.16040264, [186].log_data[56].max := 0.16079521, [186].log_data[56].total := 577.93945, [186].log_data[56].time := 3599.5, [186].log_data[56].minminute := 47, [186].log_data[56].maxminute := 5, [186].log_data[56].valid := 1, [186].log_data[57].min := 0.33655453, [186].log_data[57].max := 0.3369471, [186].log_data[57].total := 1211.9497, [186].log_data[57].time := 3599.5, [186].log_data[57].minminute := 2, [186].log_data[57].maxminute := 9, [186].log_data[57].valid := 1, [186].log_data[58].time := 3599.5, [186].log_data[58].valid := 1, [186].log_data[59].time := 3599.5, [186].log_data[59].valid := 1, [186].log_data[60].valid := 1, [186].log_data[61].valid := 1, [186].log_data[62].valid := 1, [186].log_data[63].valid := 1, [186].log_data[64].valid := 1, [186].log_data[65].valid := 1, [186].log_data[66].valid := 1, [186].log_data[67].valid := 1, [186].log_data[68].valid := 1, [186].log_data[69].valid := 1, [186].log_data[70].valid := 1, [186].log_data[71].valid := 1, [186].log_data[72].valid := 1,
        [186].log_data[73].valid := 1, [186].log_data[74].valid := 1, [186].log_data[75].valid := 1, [186].log_data[76].valid := 1, [186].log_data[77].valid := 1, [186].log_data[78].valid := 1, [186].log_data[79].valid := 1, [186].log_data[80].valid := 1, [186].log_data[81].valid := 1, [186].log_data[82].valid := 1, [186].log_data[83].valid := 1, [186].log_data[84].valid := 1, [186].log_data[85].valid := 1, [186].log_data[86].valid := 1, [186].log_data[87].valid := 1, [186].log_data[88].valid := 1, [186].log_data[89].valid := 1, [186].log_data[90].valid := 1, [186].log_data[91].valid := 1, [186].log_data[92].valid := 1, [186].log_data[93].valid := 1, [186].log_data[94].valid := 1, [186].log_data[95].valid := 1, [186].log_data[96].valid := 1, [186].log_data[97].valid := 1, [186].log_data[98].valid := 1, [186].log_data[99].valid := 1, [186].log_data[100].valid := 1, [186].log_data[101].valid := 1, [186].log_data[102].valid := 1, [186].log_data[103].valid := 1, [186].log_data[104].valid := 1, [186].log_data[105].valid := 1, [186].log_data[106].valid := 1, [186].log_data[107].valid := 1, [186].log_data[108].valid := 1, [186].log_data[109].valid := 1, [186].log_data[110].valid := 1, [186].log_data[111].valid := 1, [186].log_data[112].valid := 1, [186].log_data[113].valid := 1, [186].log_data[114].valid := 1, [186].log_data[115].valid := 1, [186].log_data[116].valid := 1, [186].log_data[117].valid := 1, [186].log_data[118].valid := 1, [186].log_data[119].valid := 1, [186].log_data[120].valid := 1, [186].log_data[121].valid := 1, [186].log_data[122].valid := 1, [186].log_data[123].valid := 1, [186].log_data[124].valid := 1, [186].time.Year := 2023, [186].time.Month := 1, [186].time.Day := 12, [186].time.Hour := 13, [186].time.Minute := 59, [186].time.Second := 59, [187].log_data[0].min := 1.0, [187].log_data[0].max := 1.0,
        [187].log_data[0].total := 3600.0, [187].log_data[0].time := 3600.0, [187].log_data[0].valid := 1, [187].log_data[1].max := 1.0, [187].log_data[1].total := 228.251, [187].log_data[1].time := 3600.0, [187].log_data[1].minminute := 3, [187].log_data[1].valid := 1, [187].log_data[2].max := 1.0, [187].log_data[2].total := 228.251, [187].log_data[2].time := 3600.0, [187].log_data[2].minminute := 3, [187].log_data[2].valid := 1, [187].log_data[3].time := 3600.0, [187].log_data[3].valid := 1, [187].log_data[4].time := 3600.0, [187].log_data[4].valid := 1, [187].log_data[5].max := 1.0, [187].log_data[5].total := 110.0, [187].log_data[5].time := 3600.0, [187].log_data[5].maxminute := 1, [187].log_data[5].valid := 1, [187].log_data[6].time := 3600.0, [187].log_data[6].valid := 1, [187].log_data[7].time := 3600.0, [187].log_data[7].valid := 1, [187].log_data[8].min := 1.0, [187].log_data[8].max := 1.0, [187].log_data[8].total := 3600.0, [187].log_data[8].time := 3600.0, [187].log_data[8].valid := 1, [187].log_data[9].min := 1.0, [187].log_data[9].max := 1.0, [187].log_data[9].total := 3600.0, [187].log_data[9].time := 3600.0, [187].log_data[9].valid := 1, [187].log_data[10].min := 1.0, [187].log_data[10].max := 1.0, [187].log_data[10].total := 3600.0, [187].log_data[10].time := 3600.0, [187].log_data[10].valid := 1, [187].log_data[11].time := 3600.0, [187].log_data[11].valid := 1, [187].log_data[12].min := 1.0, [187].log_data[12].max := 1.0, [187].log_data[12].total := 3600.0, [187].log_data[12].time := 3600.0, [187].log_data[12].valid := 1, [187].log_data[13].min := 1.0, [187].log_data[13].max := 1.0, [187].log_data[13].total := 3600.0, [187].log_data[13].time := 3600.0, [187].log_data[13].valid := 1, [187].log_data[14].time := 3600.0, [187].log_data[14].valid := 1, [187].log_data[15].time := 3600.0, [187].log_data[15].valid := 1, [187].log_data[16].time := 3600.0, [187].log_data[16].valid := 1, [187].log_data[17].min := 1.0,
        [187].log_data[17].max := 1.0, [187].log_data[17].total := 3600.0, [187].log_data[17].time := 3600.0, [187].log_data[17].valid := 1, [187].log_data[18].time := 3600.0, [187].log_data[18].valid := 1, [187].log_data[19].time := 3600.0, [187].log_data[19].valid := 1, [187].log_data[20].time := 3600.0, [187].log_data[20].valid := 1, [187].log_data[21].min := 1.0, [187].log_data[21].max := 1.0, [187].log_data[21].total := 3600.0, [187].log_data[21].time := 3600.0, [187].log_data[21].valid := 1, [187].log_data[22].time := 3600.0, [187].log_data[22].valid := 1, [187].log_data[23].time := 3600.0, [187].log_data[23].valid := 1, [187].log_data[24].time := 3600.0, [187].log_data[24].valid := 1, [187].log_data[25].time := 3600.0, [187].log_data[25].valid := 1, [187].log_data[26].time := 3600.0, [187].log_data[26].valid := 1, [187].log_data[27].time := 3600.0, [187].log_data[27].valid := 1, [187].log_data[28].time := 3600.0, [187].log_data[28].valid := 1, [187].log_data[29].min := 1.0, [187].log_data[29].max := 1.0, [187].log_data[29].total := 3600.0, [187].log_data[29].time := 3600.0, [187].log_data[29].valid := 1, [187].log_data[30].min := 1.0, [187].log_data[30].max := 1.0, [187].log_data[30].total := 3600.0, [187].log_data[30].time := 3600.0, [187].log_data[30].valid := 1, [187].log_data[31].max := 1.0, [187].log_data[31].total := 1628.7471, [187].log_data[31].time := 3600.0, [187].log_data[31].maxminute := 8, [187].log_data[31].valid := 1, [187].log_data[32].max := 1.0, [187].log_data[32].total := 1530.249, [187].log_data[32].time := 3600.0, [187].log_data[32].minminute := 7, [187].log_data[32].valid := 1, [187].log_data[33].time := 3600.0, [187].log_data[33].valid := 1, [187].log_data[34].time := 3600.0, [187].log_data[34].valid := 1, [187].log_data[35].max := 1.0, [187].log_data[35].total := 1629.7471, [187].log_data[35].time := 3600.0, [187].log_data[35].valid := 1, [187].log_data[36].max := 1.0, [187].log_data[36].total := 1469.7471, [187].log_data[36].time := 3600.0,
        [187].log_data[36].maxminute := 11, [187].log_data[36].valid := 1, [187].log_data[37].max := 6.8296957, [187].log_data[37].total := 1124.0454, [187].log_data[37].time := 3600.0, [187].log_data[37].minminute := 2, [187].log_data[37].valid := 1, [187].log_data[38].time := 3600.0, [187].log_data[38].valid := 1, [187].log_data[39].min := 0.9972973, [187].log_data[39].max := 1.0217944, [187].log_data[39].total := 3614.423, [187].log_data[39].time := 3600.0, [187].log_data[39].minminute := 56, [187].log_data[39].maxminute := 1, [187].log_data[39].valid := 1, [187].log_data[40].min := 7.560194, [187].log_data[40].max := 7.5791564, [187].log_data[40].total := 27260.762, [187].log_data[40].time := 3600.0, [187].log_data[40].minminute := 47, [187].log_data[40].maxminute := 52, [187].log_data[40].valid := 1, [187].log_data[41].min := 0.06258349, [187].log_data[41].max := 0.09850488, [187].log_data[41].total := 288.1612, [187].log_data[41].time := 3600.0, [187].log_data[41].minminute := 54, [187].log_data[41].maxminute := 6, [187].log_data[41].valid := 1, [187].log_data[42].min := 2.2929382, [187].log_data[42].max := 2.2976491, [187].log_data[42].total := 8264.025, [187].log_data[42].time := 3600.0, [187].log_data[42].minminute := 14, [187].log_data[42].maxminute := 8, [187].log_data[42].valid := 1, [187].log_data[43].min := -0.26000214, [187].log_data[43].max := -0.23999786, [187].log_data[43].total := -935.93317, [187].log_data[43].time := 3600.0, [187].log_data[43].maxminute := 8, [187].log_data[43].valid := 1, [187].log_data[44].min := -0.30000305, [187].log_data[44].max := -0.27999878, [187].log_data[44].total := -1031.8707, [187].log_data[44].time := 3600.0, [187].log_data[44].valid := 1, [187].log_data[45].time := 3600.0, [187].log_data[45].valid := 1, [187].log_data[46].time := 3600.0, [187].log_data[46].valid := 1, [187].log_data[47].time := 3600.0, [187].log_data[47].valid := 1, [187].log_data[48].min := 6.5777564, [187].log_data[48].max := 6.946274, [187].log_data[48].total := 24229.58, [187].log_data[48].time := 3600.0, [187].log_data[48].minminute := 25, [187].log_data[48].maxminute := 3,
        [187].log_data[48].valid := 1, [187].log_data[49].min := 6.675248, [187].log_data[49].max := 9.249413, [187].log_data[49].total := 28529.777, [187].log_data[49].time := 3600.0, [187].log_data[49].minminute := 22, [187].log_data[49].maxminute := 59, [187].log_data[49].valid := 1, [187].log_data[50].min := 2.0300648, [187].log_data[50].max := 2.1118004, [187].log_data[50].total := 7468.97, [187].log_data[50].time := 3600.0, [187].log_data[50].minminute := 59, [187].log_data[50].maxminute := 5, [187].log_data[50].valid := 1, [187].log_data[51].time := 3600.0, [187].log_data[51].valid := 1, [187].log_data[52].min := -2.9199982, [187].log_data[52].max := 0.13999939, [187].log_data[52].total := -7671.008, [187].log_data[52].time := 3600.0, [187].log_data[52].minminute := 8, [187].log_data[52].maxminute := 7, [187].log_data[52].valid := 1, [187].log_data[53].min := -2.4800034, [187].log_data[53].max := 0.22000122, [187].log_data[53].total := -6891.756, [187].log_data[53].time := 3600.0, [187].log_data[53].minminute := 1, [187].log_data[53].maxminute := 10, [187].log_data[53].valid := 1, [187].log_data[54].max := 0.546, [187].log_data[54].total := 1254.6321, [187].log_data[54].time := 3600.0, [187].log_data[54].minminute := 7, [187].log_data[54].maxminute := 8, [187].log_data[54].valid := 1, [187].log_data[55].max := 0.54249996, [187].log_data[55].total := 1228.7072, [187].log_data[55].time := 3600.0, [187].log_data[55].maxminute := 22, [187].log_data[55].valid := 1, [187].log_data[56].min := 0.16036338, [187].log_data[56].max := 0.16079521, [187].log_data[56].total := 577.9204, [187].log_data[56].time := 3600.0, [187].log_data[56].minminute := 15, [187].log_data[56].maxminute := 7, [187].log_data[56].valid := 1, [187].log_data[57].min := 0.33474863, [187].log_data[57].max := 0.3369471, [187].log_data[57].total := 1208.6879, [187].log_data[57].time := 3600.0, [187].log_data[57].minminute := 49, [187].log_data[57].maxminute := 10, [187].log_data[57].valid := 1, [187].log_data[58].time := 3600.0, [187].log_data[58].valid := 1, [187].log_data[59].time := 3600.0, [187].log_data[59].valid := 1,
        [187].log_data[60].valid := 1, [187].log_data[61].valid := 1, [187].log_data[62].valid := 1, [187].log_data[63].valid := 1, [187].log_data[64].valid := 1, [187].log_data[65].valid := 1, [187].log_data[66].valid := 1, [187].log_data[67].valid := 1, [187].log_data[68].valid := 1, [187].log_data[69].valid := 1, [187].log_data[70].valid := 1, [187].log_data[71].valid := 1, [187].log_data[72].valid := 1, [187].log_data[73].valid := 1, [187].log_data[74].valid := 1, [187].log_data[75].valid := 1, [187].log_data[76].valid := 1, [187].log_data[77].valid := 1, [187].log_data[78].valid := 1, [187].log_data[79].valid := 1, [187].log_data[80].valid := 1, [187].log_data[81].valid := 1, [187].log_data[82].valid := 1, [187].log_data[83].valid := 1, [187].log_data[84].valid := 1, [187].log_data[85].valid := 1, [187].log_data[86].valid := 1, [187].log_data[87].valid := 1, [187].log_data[88].valid := 1, [187].log_data[89].valid := 1, [187].log_data[90].valid := 1, [187].log_data[91].valid := 1, [187].log_data[92].valid := 1, [187].log_data[93].valid := 1, [187].log_data[94].valid := 1, [187].log_data[95].valid := 1, [187].log_data[96].valid := 1, [187].log_data[97].valid := 1, [187].log_data[98].valid := 1, [187].log_data[99].valid := 1, [187].log_data[100].valid := 1, [187].log_data[101].valid := 1, [187].log_data[102].valid := 1, [187].log_data[103].valid := 1, [187].log_data[104].valid := 1, [187].log_data[105].valid := 1, [187].log_data[106].valid := 1, [187].log_data[107].valid := 1, [187].log_data[108].valid := 1, [187].log_data[109].valid := 1, [187].log_data[110].valid := 1, [187].log_data[111].valid := 1, [187].log_data[112].valid := 1, [187].log_data[113].valid := 1, [187].log_data[114].valid := 1, [187].log_data[115].valid := 1, [187].log_data[116].valid := 1, [187].log_data[117].valid := 1, [187].log_data[118].valid := 1, [187].log_data[119].valid := 1,
        [187].log_data[120].valid := 1, [187].log_data[121].valid := 1, [187].log_data[122].valid := 1, [187].log_data[123].valid := 1, [187].log_data[124].valid := 1, [187].time.Year := 2023, [187].time.Month := 1, [187].time.Day := 12, [187].time.Hour := 14, [187].time.Minute := 59, [187].time.Second := 59, [188].log_data[0].min := 1.0, [188].log_data[0].max := 1.0, [188].log_data[0].total := 3600.0, [188].log_data[0].time := 3600.0, [188].log_data[0].valid := 1, [188].log_data[1].max := 1.0, [188].log_data[1].total := 174.249, [188].log_data[1].time := 3600.0, [188].log_data[1].maxminute := 57, [188].log_data[1].valid := 1, [188].log_data[2].max := 1.0, [188].log_data[2].total := 170.749, [188].log_data[2].time := 3600.0, [188].log_data[2].maxminute := 57, [188].log_data[2].valid := 1, [188].log_data[3].time := 3600.0, [188].log_data[3].valid := 1, [188].log_data[4].time := 3600.0, [188].log_data[4].valid := 1, [188].log_data[5].max := 1.0, [188].log_data[5].total := 40.249, [188].log_data[5].time := 3600.0, [188].log_data[5].maxminute := 59, [188].log_data[5].valid := 1, [188].log_data[6].time := 3600.0, [188].log_data[6].valid := 1, [188].log_data[7].time := 3600.0, [188].log_data[7].valid := 1, [188].log_data[8].max := 1.0, [188].log_data[8].total := 1382.751, [188].log_data[8].time := 3600.0, [188].log_data[8].minminute := 23, [188].log_data[8].valid := 1, [188].log_data[9].max := 1.0, [188].log_data[9].total := 1382.751, [188].log_data[9].time := 3600.0, [188].log_data[9].minminute := 23, [188].log_data[9].valid := 1, [188].log_data[10].min := 1.0, [188].log_data[10].max := 1.0, [188].log_data[10].total := 3600.0, [188].log_data[10].time := 3600.0, [188].log_data[10].valid := 1, [188].log_data[11].time := 3600.0, [188].log_data[11].valid := 1, [188].log_data[12].min := 1.0, [188].log_data[12].max := 1.0, [188].log_data[12].total := 3600.0, [188].log_data[12].time := 3600.0,
        [188].log_data[12].valid := 1, [188].log_data[13].min := 1.0, [188].log_data[13].max := 1.0, [188].log_data[13].total := 3600.0, [188].log_data[13].time := 3600.0, [188].log_data[13].valid := 1, [188].log_data[14].time := 3600.0, [188].log_data[14].valid := 1, [188].log_data[15].time := 3600.0, [188].log_data[15].valid := 1, [188].log_data[16].time := 3600.0, [188].log_data[16].valid := 1, [188].log_data[17].min := 1.0, [188].log_data[17].max := 1.0, [188].log_data[17].total := 3600.0, [188].log_data[17].time := 3600.0, [188].log_data[17].valid := 1, [188].log_data[18].time := 3600.0, [188].log_data[18].valid := 1, [188].log_data[19].time := 3600.0, [188].log_data[19].valid := 1, [188].log_data[20].time := 3600.0, [188].log_data[20].valid := 1, [188].log_data[21].min := 1.0, [188].log_data[21].max := 1.0, [188].log_data[21].total := 3600.0, [188].log_data[21].time := 3600.0, [188].log_data[21].valid := 1, [188].log_data[22].time := 3600.0, [188].log_data[22].valid := 1, [188].log_data[23].time := 3600.0, [188].log_data[23].valid := 1, [188].log_data[24].time := 3600.0, [188].log_data[24].valid := 1, [188].log_data[25].time := 3600.0, [188].log_data[25].valid := 1, [188].log_data[26].time := 3600.0, [188].log_data[26].valid := 1, [188].log_data[27].time := 3600.0, [188].log_data[27].valid := 1, [188].log_data[28].time := 3600.0, [188].log_data[28].valid := 1, [188].log_data[29].min := 1.0, [188].log_data[29].max := 1.0, [188].log_data[29].total := 3600.0, [188].log_data[29].time := 3600.0, [188].log_data[29].valid := 1, [188].log_data[30].min := 1.0, [188].log_data[30].max := 1.0, [188].log_data[30].total := 3600.0, [188].log_data[30].time := 3600.0, [188].log_data[30].valid := 1, [188].log_data[31].max := 1.0, [188].log_data[31].total := 544.249, [188].log_data[31].time := 3600.0, [188].log_data[31].valid := 1, [188].log_data[32].max := 1.0, [188].log_data[32].total := 577.49805, [188].log_data[32].time := 3600.0, [188].log_data[32].maxminute := 1,
        [188].log_data[32].valid := 1, [188].log_data[33].time := 3600.0, [188].log_data[33].valid := 1, [188].log_data[34].time := 3600.0, [188].log_data[34].valid := 1, [188].log_data[35].max := 1.0, [188].log_data[35].total := 543.249, [188].log_data[35].time := 3600.0, [188].log_data[35].maxminute := 4, [188].log_data[35].valid := 1, [188].log_data[36].max := 1.0, [188].log_data[36].total := 666.749, [188].log_data[36].time := 3600.0, [188].log_data[36].minminute := 2, [188].log_data[36].valid := 1, [188].log_data[37].max := 7.539878, [188].log_data[37].total := 1287.5447, [188].log_data[37].time := 3600.0, [188].log_data[37].maxminute := 58, [188].log_data[37].valid := 1, [188].log_data[38].time := 3600.0, [188].log_data[38].valid := 1, [188].log_data[39].min := 0.9982394, [188].log_data[39].max := 1.0217944, [188].log_data[39].total := 3614.2922, [188].log_data[39].time := 3600.0, [188].log_data[39].minminute := 12, [188].log_data[39].maxminute := 59, [188].log_data[39].valid := 1, [188].log_data[40].min := 7.5401335, [188].log_data[40].max := 7.592072, [188].log_data[40].total := 27255.314, [188].log_data[40].time := 3600.0, [188].log_data[40].minminute := 49, [188].log_data[40].maxminute := 53, [188].log_data[40].valid := 1, [188].log_data[41].min := 0.05944287, [188].log_data[41].max := 0.09438281, [188].log_data[41].total := 280.79657, [188].log_data[41].time := 3600.0, [188].log_data[41].minminute := 42, [188].log_data[41].maxminute := 17, [188].log_data[41].valid := 1, [188].log_data[42].min := 2.293056, [188].log_data[42].max := 2.297767, [188].log_data[42].total := 8264.124, [188].log_data[42].time := 3600.0, [188].log_data[42].minminute := 22, [188].log_data[42].maxminute := 59, [188].log_data[42].valid := 1, [188].log_data[43].min := -0.26000214, [188].log_data[43].max := -0.23999786, [188].log_data[43].total := -935.5229, [188].log_data[43].time := 3600.0, [188].log_data[43].maxminute := 19, [188].log_data[43].valid := 1, [188].log_data[44].min := -0.30000305, [188].log_data[44].max := -0.27999878, [188].log_data[44].total := -1013.5945, [188].log_data[44].time := 3600.0,
        [188].log_data[44].valid := 1, [188].log_data[45].time := 3600.0, [188].log_data[45].valid := 1, [188].log_data[46].time := 3600.0, [188].log_data[46].valid := 1, [188].log_data[47].time := 3600.0, [188].log_data[47].valid := 1, [188].log_data[48].min := 6.7506104, [188].log_data[48].max := 6.795404, [188].log_data[48].total := 24316.025, [188].log_data[48].time := 3600.0, [188].log_data[48].minminute := 24, [188].log_data[48].maxminute := 59, [188].log_data[48].valid := 1, [188].log_data[49].min := 9.238029, [188].log_data[49].max := 9.372684, [188].log_data[49].total := 33619.27, [188].log_data[49].time := 3600.0, [188].log_data[49].maxminute := 25, [188].log_data[49].valid := 1, [188].log_data[50].min := 1.9994433, [188].log_data[50].max := 2.1269934, [188].log_data[50].total := 7451.5996, [188].log_data[50].time := 3600.0, [188].log_data[50].minminute := 23, [188].log_data[50].maxminute := 59, [188].log_data[50].valid := 1, [188].log_data[51].time := 3600.0, [188].log_data[51].valid := 1, [188].log_data[52].min := -2.7600021, [188].log_data[52].max := 0.13999939, [188].log_data[52].total := -5756.777, [188].log_data[52].time := 3600.0, [188].log_data[52].minminute := 12, [188].log_data[52].valid := 1, [188].log_data[53].min := -2.4800034, [188].log_data[53].max := 0.22000122, [188].log_data[53].total := -5637.936, [188].log_data[53].time := 3600.0, [188].log_data[53].minminute := 10, [188].log_data[53].maxminute := 4, [188].log_data[53].valid := 1, [188].log_data[54].max := 0.507, [188].log_data[54].total := 443.65125, [188].log_data[54].time := 3600.0, [188].log_data[54].maxminute := 12, [188].log_data[54].valid := 1, [188].log_data[55].max := 0.50299996, [188].log_data[55].total := 480.88495, [188].log_data[55].time := 3600.0, [188].log_data[55].minminute := 2, [188].log_data[55].maxminute := 14, [188].log_data[55].valid := 1, [188].log_data[56].min := 0.16032413, [188].log_data[56].max := 0.1607167, [188].log_data[56].total := 577.8123, [188].log_data[56].time := 3600.0, [188].log_data[56].minminute := 36, [188].log_data[56].maxminute := 1, [188].log_data[56].valid := 1,
        [188].log_data[57].min := 0.3347879, [188].log_data[57].max := 0.33521977, [188].log_data[57].total := 1205.8947, [188].log_data[57].time := 3600.0, [188].log_data[57].maxminute := 29, [188].log_data[57].valid := 1, [188].log_data[58].time := 3600.0, [188].log_data[58].valid := 1, [188].log_data[59].time := 3600.0, [188].log_data[59].valid := 1, [188].log_data[60].valid := 1, [188].log_data[61].valid := 1, [188].log_data[62].valid := 1, [188].log_data[63].valid := 1, [188].log_data[64].valid := 1, [188].log_data[65].valid := 1, [188].log_data[66].valid := 1, [188].log_data[67].valid := 1, [188].log_data[68].valid := 1, [188].log_data[69].valid := 1, [188].log_data[70].valid := 1, [188].log_data[71].valid := 1, [188].log_data[72].valid := 1, [188].log_data[73].valid := 1, [188].log_data[74].valid := 1, [188].log_data[75].valid := 1, [188].log_data[76].valid := 1, [188].log_data[77].valid := 1, [188].log_data[78].valid := 1, [188].log_data[79].valid := 1, [188].log_data[80].valid := 1, [188].log_data[81].valid := 1, [188].log_data[82].valid := 1, [188].log_data[83].valid := 1, [188].log_data[84].valid := 1, [188].log_data[85].valid := 1, [188].log_data[86].valid := 1, [188].log_data[87].valid := 1, [188].log_data[88].valid := 1, [188].log_data[89].valid := 1, [188].log_data[90].valid := 1, [188].log_data[91].valid := 1, [188].log_data[92].valid := 1, [188].log_data[93].valid := 1, [188].log_data[94].valid := 1, [188].log_data[95].valid := 1, [188].log_data[96].valid := 1, [188].log_data[97].valid := 1, [188].log_data[98].valid := 1, [188].log_data[99].valid := 1, [188].log_data[100].valid := 1, [188].log_data[101].valid := 1, [188].log_data[102].valid := 1, [188].log_data[103].valid := 1, [188].log_data[104].valid := 1, [188].log_data[105].valid := 1, [188].log_data[106].valid := 1, [188].log_data[107].valid := 1, [188].log_data[108].valid := 1, [188].log_data[109].valid := 1,
        [188].log_data[110].valid := 1, [188].log_data[111].valid := 1, [188].log_data[112].valid := 1, [188].log_data[113].valid := 1, [188].log_data[114].valid := 1, [188].log_data[115].valid := 1, [188].log_data[116].valid := 1, [188].log_data[117].valid := 1, [188].log_data[118].valid := 1, [188].log_data[119].valid := 1, [188].log_data[120].valid := 1, [188].log_data[121].valid := 1, [188].log_data[122].valid := 1, [188].log_data[123].valid := 1, [188].log_data[124].valid := 1, [188].time.Year := 2023, [188].time.Month := 1, [188].time.Day := 12, [188].time.Hour := 15, [188].time.Minute := 59, [188].time.Second := 59, [189].log_data[0].min := 1.0, [189].log_data[0].max := 1.0, [189].log_data[0].total := 3600.0, [189].log_data[0].time := 3600.0, [189].log_data[0].valid := 1, [189].log_data[1].max := 1.0, [189].log_data[1].total := 357.751, [189].log_data[1].time := 3600.0, [189].log_data[1].minminute := 5, [189].log_data[1].valid := 1, [189].log_data[2].max := 1.0, [189].log_data[2].total := 357.751, [189].log_data[2].time := 3600.0, [189].log_data[2].minminute := 5, [189].log_data[2].valid := 1, [189].log_data[3].time := 3600.0, [189].log_data[3].valid := 1, [189].log_data[4].time := 3600.0, [189].log_data[4].valid := 1, [189].log_data[5].max := 1.0, [189].log_data[5].total := 203.251, [189].log_data[5].time := 3600.0, [189].log_data[5].minminute := 1, [189].log_data[5].valid := 1, [189].log_data[6].time := 3600.0, [189].log_data[6].valid := 1, [189].log_data[7].time := 3600.0, [189].log_data[7].valid := 1, [189].log_data[8].max := 1.0, [189].log_data[8].total := 3549.749, [189].log_data[8].time := 3600.0, [189].log_data[8].valid := 1, [189].log_data[9].max := 1.0, [189].log_data[9].total := 3546.249, [189].log_data[9].time := 3600.0, [189].log_data[9].valid := 1, [189].log_data[10].min := 1.0, [189].log_data[10].max := 1.0, [189].log_data[10].total := 3600.0,
        [189].log_data[10].time := 3600.0, [189].log_data[10].valid := 1, [189].log_data[11].time := 3600.0, [189].log_data[11].valid := 1, [189].log_data[12].min := 1.0, [189].log_data[12].max := 1.0, [189].log_data[12].total := 3600.0, [189].log_data[12].time := 3600.0, [189].log_data[12].valid := 1, [189].log_data[13].min := 1.0, [189].log_data[13].max := 1.0, [189].log_data[13].total := 3600.0, [189].log_data[13].time := 3600.0, [189].log_data[13].valid := 1, [189].log_data[14].time := 3600.0, [189].log_data[14].valid := 1, [189].log_data[15].time := 3600.0, [189].log_data[15].valid := 1, [189].log_data[16].time := 3600.0, [189].log_data[16].valid := 1, [189].log_data[17].min := 1.0, [189].log_data[17].max := 1.0, [189].log_data[17].total := 3600.0, [189].log_data[17].time := 3600.0, [189].log_data[17].valid := 1, [189].log_data[18].time := 3600.0, [189].log_data[18].valid := 1, [189].log_data[19].time := 3600.0, [189].log_data[19].valid := 1, [189].log_data[20].time := 3600.0, [189].log_data[20].valid := 1, [189].log_data[21].min := 1.0, [189].log_data[21].max := 1.0, [189].log_data[21].total := 3600.0, [189].log_data[21].time := 3600.0, [189].log_data[21].valid := 1, [189].log_data[22].time := 3600.0, [189].log_data[22].valid := 1, [189].log_data[23].time := 3600.0, [189].log_data[23].valid := 1, [189].log_data[24].time := 3600.0, [189].log_data[24].valid := 1, [189].log_data[25].time := 3600.0, [189].log_data[25].valid := 1, [189].log_data[26].time := 3600.0, [189].log_data[26].valid := 1, [189].log_data[27].time := 3600.0, [189].log_data[27].valid := 1, [189].log_data[28].time := 3600.0, [189].log_data[28].valid := 1, [189].log_data[29].min := 1.0, [189].log_data[29].max := 1.0, [189].log_data[29].total := 3600.0, [189].log_data[29].time := 3600.0, [189].log_data[29].valid := 1, [189].log_data[30].min := 1.0, [189].log_data[30].max := 1.0, [189].log_data[30].total := 3600.0, [189].log_data[30].time := 3600.0, [189].log_data[30].valid := 1,
        [189].log_data[31].max := 1.0, [189].log_data[31].total := 1595.2471, [189].log_data[31].time := 3600.0, [189].log_data[31].valid := 1, [189].log_data[32].max := 1.0, [189].log_data[32].total := 1506.498, [189].log_data[32].time := 3600.0, [189].log_data[32].maxminute := 10, [189].log_data[32].valid := 1, [189].log_data[33].time := 3600.0, [189].log_data[33].valid := 1, [189].log_data[34].time := 3600.0, [189].log_data[34].valid := 1, [189].log_data[35].max := 1.0, [189].log_data[35].total := 1379.996, [189].log_data[35].time := 3600.0, [189].log_data[35].maxminute := 1, [189].log_data[35].valid := 1, [189].log_data[36].max := 1.0, [189].log_data[36].total := 1629.7471, [189].log_data[36].time := 3600.0, [189].log_data[36].maxminute := 3, [189].log_data[36].valid := 1, [189].log_data[37].max := 7.461754, [189].log_data[37].total := 2174.5112, [189].log_data[37].time := 3600.0, [189].log_data[37].minminute := 4, [189].log_data[37].valid := 1, [189].log_data[38].time := 3600.0, [189].log_data[38].valid := 1, [189].log_data[39].min := 0.99423516, [189].log_data[39].max := 1.0221478, [189].log_data[39].total := 3604.4575, [189].log_data[39].time := 3600.0, [189].log_data[39].minminute := 43, [189].log_data[39].maxminute := 3, [189].log_data[39].valid := 1, [189].log_data[40].min := 7.5486526, [189].log_data[40].max := 7.584652, [189].log_data[40].total := 27253.963, [189].log_data[40].time := 3600.0, [189].log_data[40].minminute := 22, [189].log_data[40].maxminute := 36, [189].log_data[40].valid := 1, [189].log_data[41].min := 0.04727295, [189].log_data[41].max := 0.08829786, [189].log_data[41].total := 231.81345, [189].log_data[41].time := 3600.0, [189].log_data[41].minminute := 52, [189].log_data[41].maxminute := 31, [189].log_data[41].valid := 1, [189].log_data[42].min := 2.2929382, [189].log_data[42].max := 2.297767, [189].log_data[42].total := 8264.15, [189].log_data[42].time := 3600.0, [189].log_data[42].minminute := 15, [189].log_data[42].maxminute := 39, [189].log_data[42].valid := 1, [189].log_data[43].min := -0.26000214, [189].log_data[43].max := -0.23999786,
        [189].log_data[43].total := -935.4082, [189].log_data[43].time := 3600.0, [189].log_data[43].valid := 1, [189].log_data[44].min := -0.30000305, [189].log_data[44].max := -0.27999878, [189].log_data[44].total := -1008.6443, [189].log_data[44].time := 3600.0, [189].log_data[44].valid := 1, [189].log_data[45].time := 3600.0, [189].log_data[45].valid := 1, [189].log_data[46].time := 3600.0, [189].log_data[46].valid := 1, [189].log_data[47].time := 3600.0, [189].log_data[47].valid := 1, [189].log_data[48].min := 6.58655, [189].log_data[48].max := 6.9465485, [189].log_data[48].total := 24261.43, [189].log_data[48].time := 3600.0, [189].log_data[48].minminute := 28, [189].log_data[48].maxminute := 6, [189].log_data[48].valid := 1, [189].log_data[49].min := 6.638737, [189].log_data[49].max := 9.342062, [189].log_data[49].total := 28459.848, [189].log_data[49].time := 3600.0, [189].log_data[49].minminute := 26, [189].log_data[49].valid := 1, [189].log_data[50].min := 2.0438442, [189].log_data[50].max := 2.150784, [189].log_data[50].total := 7505.209, [189].log_data[50].time := 3600.0, [189].log_data[50].minminute := 59, [189].log_data[50].valid := 1, [189].log_data[51].time := 3600.0, [189].log_data[51].valid := 1, [189].log_data[52].min := -4.1399994, [189].log_data[52].max := 0.13999939, [189].log_data[52].total := -7663.1147, [189].log_data[52].time := 3600.0, [189].log_data[52].minminute := 1, [189].log_data[52].maxminute := 30, [189].log_data[52].valid := 1, [189].log_data[53].min := -3.8399963, [189].log_data[53].max := 0.22000122, [189].log_data[53].total := -6865.4937, [189].log_data[53].time := 3600.0, [189].log_data[53].minminute := 1, [189].log_data[53].maxminute := 12, [189].log_data[53].valid := 1, [189].log_data[54].max := 0.543, [189].log_data[54].total := 1229.2816, [189].log_data[54].time := 3600.0, [189].log_data[54].maxminute := 42, [189].log_data[54].valid := 1, [189].log_data[55].max := 0.537, [189].log_data[55].total := 1190.4376, [189].log_data[55].time := 3600.0, [189].log_data[55].maxminute := 13, [189].log_data[55].valid := 1, [189].log_data[56].min := 0.16028486,
        [189].log_data[56].max := 0.1607167, [189].log_data[56].total := 577.70795, [189].log_data[56].time := 3600.0, [189].log_data[56].minminute := 23, [189].log_data[56].maxminute := 10, [189].log_data[56].valid := 1, [189].log_data[57].min := 0.33337462, [189].log_data[57].max := 0.33521977, [189].log_data[57].total := 1203.4122, [189].log_data[57].time := 3600.0, [189].log_data[57].minminute := 37, [189].log_data[57].maxminute := 15, [189].log_data[57].valid := 1, [189].log_data[58].time := 3600.0, [189].log_data[58].valid := 1, [189].log_data[59].time := 3600.0, [189].log_data[59].valid := 1, [189].log_data[60].valid := 1, [189].log_data[61].valid := 1, [189].log_data[62].valid := 1, [189].log_data[63].valid := 1, [189].log_data[64].valid := 1, [189].log_data[65].valid := 1, [189].log_data[66].valid := 1, [189].log_data[67].valid := 1, [189].log_data[68].valid := 1, [189].log_data[69].valid := 1, [189].log_data[70].valid := 1, [189].log_data[71].valid := 1, [189].log_data[72].valid := 1, [189].log_data[73].valid := 1, [189].log_data[74].valid := 1, [189].log_data[75].valid := 1, [189].log_data[76].valid := 1, [189].log_data[77].valid := 1, [189].log_data[78].valid := 1, [189].log_data[79].valid := 1, [189].log_data[80].valid := 1, [189].log_data[81].valid := 1, [189].log_data[82].valid := 1, [189].log_data[83].valid := 1, [189].log_data[84].valid := 1, [189].log_data[85].valid := 1, [189].log_data[86].valid := 1, [189].log_data[87].valid := 1, [189].log_data[88].valid := 1, [189].log_data[89].valid := 1, [189].log_data[90].valid := 1, [189].log_data[91].valid := 1, [189].log_data[92].valid := 1, [189].log_data[93].valid := 1, [189].log_data[94].valid := 1, [189].log_data[95].valid := 1, [189].log_data[96].valid := 1, [189].log_data[97].valid := 1, [189].log_data[98].valid := 1, [189].log_data[99].valid := 1, [189].log_data[100].valid := 1, [189].log_data[101].valid := 1, [189].log_data[102].valid := 1,
        [189].log_data[103].valid := 1, [189].log_data[104].valid := 1, [189].log_data[105].valid := 1, [189].log_data[106].valid := 1, [189].log_data[107].valid := 1, [189].log_data[108].valid := 1, [189].log_data[109].valid := 1, [189].log_data[110].valid := 1, [189].log_data[111].valid := 1, [189].log_data[112].valid := 1, [189].log_data[113].valid := 1, [189].log_data[114].valid := 1, [189].log_data[115].valid := 1, [189].log_data[116].valid := 1, [189].log_data[117].valid := 1, [189].log_data[118].valid := 1, [189].log_data[119].valid := 1, [189].log_data[120].valid := 1, [189].log_data[121].valid := 1, [189].log_data[122].valid := 1, [189].log_data[123].valid := 1, [189].log_data[124].valid := 1, [189].time.Year := 2023, [189].time.Month := 1, [189].time.Day := 12, [189].time.Hour := 16, [189].time.Minute := 59, [189].time.Second := 59, [190].log_data[0].min := 1.0, [190].log_data[0].max := 1.0, [190].log_data[0].total := 3600.0, [190].log_data[0].time := 3600.0, [190].log_data[0].valid := 1, [190].log_data[1].max := 1.0, [190].log_data[1].total := 587.0, [190].log_data[1].time := 3600.0, [190].log_data[1].maxminute := 22, [190].log_data[1].valid := 1, [190].log_data[2].max := 1.0, [190].log_data[2].total := 583.5, [190].log_data[2].time := 3600.0, [190].log_data[2].maxminute := 22, [190].log_data[2].valid := 1, [190].log_data[3].time := 3600.0, [190].log_data[3].valid := 1, [190].log_data[4].time := 3600.0, [190].log_data[4].valid := 1, [190].log_data[5].max := 1.0, [190].log_data[5].total := 231.0, [190].log_data[5].time := 3600.0, [190].log_data[5].maxminute := 24, [190].log_data[5].valid := 1, [190].log_data[6].time := 3600.0, [190].log_data[6].valid := 1, [190].log_data[7].time := 3600.0, [190].log_data[7].valid := 1, [190].log_data[8].min := 1.0, [190].log_data[8].max := 1.0, [190].log_data[8].total := 3600.0, [190].log_data[8].time := 3600.0,
        [190].log_data[8].valid := 1, [190].log_data[9].min := 1.0, [190].log_data[9].max := 1.0, [190].log_data[9].total := 3600.0, [190].log_data[9].time := 3600.0, [190].log_data[9].valid := 1, [190].log_data[10].min := 1.0, [190].log_data[10].max := 1.0, [190].log_data[10].total := 3600.0, [190].log_data[10].time := 3600.0, [190].log_data[10].valid := 1, [190].log_data[11].time := 3600.0, [190].log_data[11].valid := 1, [190].log_data[12].min := 1.0, [190].log_data[12].max := 1.0, [190].log_data[12].total := 3600.0, [190].log_data[12].time := 3600.0, [190].log_data[12].valid := 1, [190].log_data[13].min := 1.0, [190].log_data[13].max := 1.0, [190].log_data[13].total := 3600.0, [190].log_data[13].time := 3600.0, [190].log_data[13].valid := 1, [190].log_data[14].time := 3600.0, [190].log_data[14].valid := 1, [190].log_data[15].time := 3600.0, [190].log_data[15].valid := 1, [190].log_data[16].time := 3600.0, [190].log_data[16].valid := 1, [190].log_data[17].min := 1.0, [190].log_data[17].max := 1.0, [190].log_data[17].total := 3600.0, [190].log_data[17].time := 3600.0, [190].log_data[17].valid := 1, [190].log_data[18].time := 3600.0, [190].log_data[18].valid := 1, [190].log_data[19].time := 3600.0, [190].log_data[19].valid := 1, [190].log_data[20].time := 3600.0, [190].log_data[20].valid := 1, [190].log_data[21].min := 1.0, [190].log_data[21].max := 1.0, [190].log_data[21].total := 3600.0, [190].log_data[21].time := 3600.0, [190].log_data[21].valid := 1, [190].log_data[22].time := 3600.0, [190].log_data[22].valid := 1, [190].log_data[23].time := 3600.0, [190].log_data[23].valid := 1, [190].log_data[24].time := 3600.0, [190].log_data[24].valid := 1, [190].log_data[25].time := 3600.0, [190].log_data[25].valid := 1, [190].log_data[26].time := 3600.0, [190].log_data[26].valid := 1, [190].log_data[27].time := 3600.0, [190].log_data[27].valid := 1, [190].log_data[28].time := 3600.0, [190].log_data[28].valid := 1, [190].log_data[29].min := 1.0,
        [190].log_data[29].max := 1.0, [190].log_data[29].total := 3600.0, [190].log_data[29].time := 3600.0, [190].log_data[29].valid := 1, [190].log_data[30].min := 1.0, [190].log_data[30].max := 1.0, [190].log_data[30].total := 3600.0, [190].log_data[30].time := 3600.0, [190].log_data[30].valid := 1, [190].log_data[31].max := 1.0, [190].log_data[31].total := 1629.998, [190].log_data[31].time := 3600.0, [190].log_data[31].maxminute := 3, [190].log_data[31].valid := 1, [190].log_data[32].max := 1.0, [190].log_data[32].total := 1440.2471, [190].log_data[32].time := 3600.0, [190].log_data[32].minminute := 2, [190].log_data[32].valid := 1, [190].log_data[33].time := 3600.0, [190].log_data[33].valid := 1, [190].log_data[34].time := 3600.0, [190].log_data[34].valid := 1, [190].log_data[35].max := 1.0, [190].log_data[35].total := 1440.498, [190].log_data[35].time := 3600.0, [190].log_data[35].minminute := 4, [190].log_data[35].valid := 1, [190].log_data[36].max := 1.0, [190].log_data[36].total := 1629.998, [190].log_data[36].time := 3600.0, [190].log_data[36].maxminute := 6, [190].log_data[36].valid := 1, [190].log_data[37].max := 6.999684, [190].log_data[37].total := 3578.1191, [190].log_data[37].time := 3600.0, [190].log_data[37].maxminute := 25, [190].log_data[37].valid := 1, [190].log_data[38].time := 3600.0, [190].log_data[38].valid := 1, [190].log_data[39].min := 0.9936463, [190].log_data[39].max := 1.0208522, [190].log_data[39].total := 3610.8198, [190].log_data[39].time := 3600.0, [190].log_data[39].minminute := 22, [190].log_data[39].maxminute := 24, [190].log_data[39].valid := 1, [190].log_data[40].min := 7.550027, [190].log_data[40].max := 7.590423, [190].log_data[40].total := 27261.262, [190].log_data[40].time := 3600.0, [190].log_data[40].minminute := 22, [190].log_data[40].maxminute := 30, [190].log_data[40].valid := 1, [190].log_data[41].min := 0.050217286, [190].log_data[41].max := 0.08613843, [190].log_data[41].total := 247.54936, [190].log_data[41].time := 3600.0, [190].log_data[41].maxminute := 49, [190].log_data[41].valid := 1,
        [190].log_data[42].min := 2.2928205, [190].log_data[42].max := 2.2976491, [190].log_data[42].total := 8264.192, [190].log_data[42].time := 3600.0, [190].log_data[42].minminute := 24, [190].log_data[42].maxminute := 5, [190].log_data[42].valid := 1, [190].log_data[43].min := -0.26000214, [190].log_data[43].max := -0.23999786, [190].log_data[43].total := -935.9482, [190].log_data[43].time := 3600.0, [190].log_data[43].maxminute := 5, [190].log_data[43].valid := 1, [190].log_data[44].min := -0.30000305, [190].log_data[44].max := -0.27999878, [190].log_data[44].total := -1017.49994, [190].log_data[44].time := 3600.0, [190].log_data[44].valid := 1, [190].log_data[45].time := 3600.0, [190].log_data[45].valid := 1, [190].log_data[46].time := 3600.0, [190].log_data[46].valid := 1, [190].log_data[47].time := 3600.0, [190].log_data[47].valid := 1, [190].log_data[48].min := 6.57968, [190].log_data[48].max := 6.9465485, [190].log_data[48].total := 24214.553, [190].log_data[48].time := 3600.0, [190].log_data[48].minminute := 53, [190].log_data[48].maxminute := 31, [190].log_data[48].valid := 1, [190].log_data[49].min := 6.730406, [190].log_data[49].max := 9.362476, [190].log_data[49].total := 29692.719, [190].log_data[49].time := 3600.0, [190].log_data[49].minminute := 53, [190].log_data[49].maxminute := 25, [190].log_data[49].valid := 1, [190].log_data[50].min := 2.0089831, [190].log_data[50].max := 2.1146271, [190].log_data[50].total := 7436.174, [190].log_data[50].time := 3600.0, [190].log_data[50].minminute := 24, [190].log_data[50].maxminute := 31, [190].log_data[50].valid := 1, [190].log_data[51].time := 3600.0, [190].log_data[51].valid := 1, [190].log_data[52].min := -2.840004, [190].log_data[52].max := 0.13999939, [190].log_data[52].total := -7440.147, [190].log_data[52].time := 3600.0, [190].log_data[52].minminute := 14, [190].log_data[52].maxminute := 2, [190].log_data[52].valid := 1, [190].log_data[53].min := -2.4800034, [190].log_data[53].max := 0.22000122, [190].log_data[53].total := -6938.142, [190].log_data[53].time := 3600.0, [190].log_data[53].minminute := 17, [190].log_data[53].maxminute := 37,
        [190].log_data[53].valid := 1, [190].log_data[54].max := 0.5285, [190].log_data[54].total := 1216.9943, [190].log_data[54].time := 3600.0, [190].log_data[54].minminute := 2, [190].log_data[54].maxminute := 14, [190].log_data[54].valid := 1, [190].log_data[55].max := 0.518, [190].log_data[55].total := 1217.2986, [190].log_data[55].time := 3600.0, [190].log_data[55].minminute := 4, [190].log_data[55].maxminute := 6, [190].log_data[55].valid := 1, [190].log_data[56].min := 0.16028486, [190].log_data[56].max := 0.16075596, [190].log_data[56].total := 577.67957, [190].log_data[56].time := 3600.0, [190].log_data[56].minminute := 49, [190].log_data[56].maxminute := 3, [190].log_data[56].valid := 1, [190].log_data[57].min := 0.3320791, [190].log_data[57].max := 0.33372793, [190].log_data[57].total := 1200.0444, [190].log_data[57].time := 3600.0, [190].log_data[57].minminute := 59, [190].log_data[57].maxminute := 44, [190].log_data[57].valid := 1, [190].log_data[58].time := 3600.0, [190].log_data[58].valid := 1, [190].log_data[59].time := 3600.0, [190].log_data[59].valid := 1, [190].log_data[60].valid := 1, [190].log_data[61].valid := 1, [190].log_data[62].valid := 1, [190].log_data[63].valid := 1, [190].log_data[64].valid := 1, [190].log_data[65].valid := 1, [190].log_data[66].valid := 1, [190].log_data[67].valid := 1, [190].log_data[68].valid := 1, [190].log_data[69].valid := 1, [190].log_data[70].valid := 1, [190].log_data[71].valid := 1, [190].log_data[72].valid := 1, [190].log_data[73].valid := 1, [190].log_data[74].valid := 1, [190].log_data[75].valid := 1, [190].log_data[76].valid := 1, [190].log_data[77].valid := 1, [190].log_data[78].valid := 1, [190].log_data[79].valid := 1, [190].log_data[80].valid := 1, [190].log_data[81].valid := 1, [190].log_data[82].valid := 1, [190].log_data[83].valid := 1, [190].log_data[84].valid := 1, [190].log_data[85].valid := 1, [190].log_data[86].valid := 1, [190].log_data[87].valid := 1, [190].log_data[88].valid := 1,
        [190].log_data[89].valid := 1, [190].log_data[90].valid := 1, [190].log_data[91].valid := 1, [190].log_data[92].valid := 1, [190].log_data[93].valid := 1, [190].log_data[94].valid := 1, [190].log_data[95].valid := 1, [190].log_data[96].valid := 1, [190].log_data[97].valid := 1, [190].log_data[98].valid := 1, [190].log_data[99].valid := 1, [190].log_data[100].valid := 1, [190].log_data[101].valid := 1, [190].log_data[102].valid := 1, [190].log_data[103].valid := 1, [190].log_data[104].valid := 1, [190].log_data[105].valid := 1, [190].log_data[106].valid := 1, [190].log_data[107].valid := 1, [190].log_data[108].valid := 1, [190].log_data[109].valid := 1, [190].log_data[110].valid := 1, [190].log_data[111].valid := 1, [190].log_data[112].valid := 1, [190].log_data[113].valid := 1, [190].log_data[114].valid := 1, [190].log_data[115].valid := 1, [190].log_data[116].valid := 1, [190].log_data[117].valid := 1, [190].log_data[118].valid := 1, [190].log_data[119].valid := 1, [190].log_data[120].valid := 1, [190].log_data[121].valid := 1, [190].log_data[122].valid := 1, [190].log_data[123].valid := 1, [190].log_data[124].valid := 1, [190].time.Year := 2023, [190].time.Month := 1, [190].time.Day := 12, [190].time.Hour := 17, [190].time.Minute := 59, [190].time.Second := 59, [191].log_data[0].min := 1.0, [191].log_data[0].max := 1.0, [191].log_data[0].total := 3600.0, [191].log_data[0].time := 3600.0, [191].log_data[0].valid := 1, [191].log_data[1].max := 1.0, [191].log_data[1].total := 73.749, [191].log_data[1].time := 3600.0, [191].log_data[1].maxminute := 58, [191].log_data[1].valid := 1, [191].log_data[2].max := 1.0, [191].log_data[2].total := 70.249, [191].log_data[2].time := 3600.0, [191].log_data[2].maxminute := 58, [191].log_data[2].valid := 1, [191].log_data[3].time := 3600.0, [191].log_data[3].valid := 1, [191].log_data[4].time := 3600.0,
        [191].log_data[4].valid := 1, [191].log_data[5].time := 3600.0, [191].log_data[5].valid := 1, [191].log_data[6].time := 3600.0, [191].log_data[6].valid := 1, [191].log_data[7].time := 3600.0, [191].log_data[7].valid := 1, [191].log_data[8].max := 1.0, [191].log_data[8].total := 3405.751, [191].log_data[8].time := 3600.0, [191].log_data[8].minminute := 56, [191].log_data[8].valid := 1, [191].log_data[9].max := 1.0, [191].log_data[9].total := 3405.751, [191].log_data[9].time := 3600.0, [191].log_data[9].minminute := 56, [191].log_data[9].valid := 1, [191].log_data[10].min := 1.0, [191].log_data[10].max := 1.0, [191].log_data[10].total := 3600.0, [191].log_data[10].time := 3600.0, [191].log_data[10].valid := 1, [191].log_data[11].time := 3600.0, [191].log_data[11].valid := 1, [191].log_data[12].min := 1.0, [191].log_data[12].max := 1.0, [191].log_data[12].total := 3600.0, [191].log_data[12].time := 3600.0, [191].log_data[12].valid := 1, [191].log_data[13].min := 1.0, [191].log_data[13].max := 1.0, [191].log_data[13].total := 3600.0, [191].log_data[13].time := 3600.0, [191].log_data[13].valid := 1, [191].log_data[14].time := 3600.0, [191].log_data[14].valid := 1, [191].log_data[15].time := 3600.0, [191].log_data[15].valid := 1, [191].log_data[16].time := 3600.0, [191].log_data[16].valid := 1, [191].log_data[17].min := 1.0, [191].log_data[17].max := 1.0, [191].log_data[17].total := 3600.0, [191].log_data[17].time := 3600.0, [191].log_data[17].valid := 1, [191].log_data[18].time := 3600.0, [191].log_data[18].valid := 1, [191].log_data[19].time := 3600.0, [191].log_data[19].valid := 1, [191].log_data[20].time := 3600.0, [191].log_data[20].valid := 1, [191].log_data[21].min := 1.0, [191].log_data[21].max := 1.0, [191].log_data[21].total := 3600.0, [191].log_data[21].time := 3600.0, [191].log_data[21].valid := 1, [191].log_data[22].time := 3600.0, [191].log_data[22].valid := 1, [191].log_data[23].time := 3600.0, [191].log_data[23].valid := 1,
        [191].log_data[24].time := 3600.0, [191].log_data[24].valid := 1, [191].log_data[25].time := 3600.0, [191].log_data[25].valid := 1, [191].log_data[26].time := 3600.0, [191].log_data[26].valid := 1, [191].log_data[27].time := 3600.0, [191].log_data[27].valid := 1, [191].log_data[28].time := 3600.0, [191].log_data[28].valid := 1, [191].log_data[29].min := 1.0, [191].log_data[29].max := 1.0, [191].log_data[29].total := 3600.0, [191].log_data[29].time := 3600.0, [191].log_data[29].valid := 1, [191].log_data[30].min := 1.0, [191].log_data[30].max := 1.0, [191].log_data[30].total := 3600.0, [191].log_data[30].time := 3600.0, [191].log_data[30].valid := 1, [191].log_data[31].max := 1.0, [191].log_data[31].total := 1569.249, [191].log_data[31].time := 3600.0, [191].log_data[31].maxminute := 6, [191].log_data[31].valid := 1, [191].log_data[32].max := 1.0, [191].log_data[32].total := 1399.749, [191].log_data[32].time := 3600.0, [191].log_data[32].minminute := 5, [191].log_data[32].valid := 1, [191].log_data[33].time := 3600.0, [191].log_data[33].valid := 1, [191].log_data[34].time := 3600.0, [191].log_data[34].valid := 1, [191].log_data[35].max := 1.0, [191].log_data[35].total := 1561.251, [191].log_data[35].time := 3600.0, [191].log_data[35].minminute := 7, [191].log_data[35].valid := 1, [191].log_data[36].max := 1.0, [191].log_data[36].total := 1406.7471, [191].log_data[36].time := 3600.0, [191].log_data[36].maxminute := 9, [191].log_data[36].valid := 1, [191].log_data[37].max := 7.6501937, [191].log_data[37].total := 542.123, [191].log_data[37].time := 3600.0, [191].log_data[37].maxminute := 59, [191].log_data[37].valid := 1, [191].log_data[38].time := 3600.0, [191].log_data[38].valid := 1, [191].log_data[39].min := 0.99753284, [191].log_data[39].max := 1.0126079, [191].log_data[39].total := 3612.4646, [191].log_data[39].time := 3600.0, [191].log_data[39].minminute := 47, [191].log_data[39].maxminute := 59, [191].log_data[39].valid := 1, [191].log_data[40].min := 7.54453, [191].log_data[40].max := 7.587675,
        [191].log_data[40].total := 27261.824, [191].log_data[40].time := 3600.0, [191].log_data[40].minminute := 42, [191].log_data[40].maxminute := 52, [191].log_data[40].valid := 1, [191].log_data[41].min := 0.06965014, [191].log_data[41].max := 0.111656494, [191].log_data[41].total := 348.3074, [191].log_data[41].time := 3600.0, [191].log_data[41].minminute := 3, [191].log_data[41].maxminute := 19, [191].log_data[41].valid := 1, [191].log_data[42].min := 2.293056, [191].log_data[42].max := 2.297767, [191].log_data[42].total := 8264.019, [191].log_data[42].time := 3600.0, [191].log_data[42].maxminute := 7, [191].log_data[42].valid := 1, [191].log_data[43].min := -0.26000214, [191].log_data[43].max := -0.23999786, [191].log_data[43].total := -935.92816, [191].log_data[43].time := 3600.0, [191].log_data[43].maxminute := 21, [191].log_data[43].valid := 1, [191].log_data[44].min := -0.30000305, [191].log_data[44].max := -0.27999878, [191].log_data[44].total := -1015.3162, [191].log_data[44].time := 3600.0, [191].log_data[44].valid := 1, [191].log_data[45].time := 3600.0, [191].log_data[45].valid := 1, [191].log_data[46].time := 3600.0, [191].log_data[46].valid := 1, [191].log_data[47].time := 3600.0, [191].log_data[47].valid := 1, [191].log_data[48].min := 6.68768, [191].log_data[48].max := 6.7981515, [191].log_data[48].total := 24349.01, [191].log_data[48].time := 3600.0, [191].log_data[48].maxminute := 7, [191].log_data[48].valid := 1, [191].log_data[49].min := 7.571711, [191].log_data[49].max := 9.359533, [191].log_data[49].total := 32476.084, [191].log_data[49].time := 3600.0, [191].log_data[49].maxminute := 57, [191].log_data[49].valid := 1, [191].log_data[50].min := 1.9994433, [191].log_data[50].max := 2.0825925, [191].log_data[50].total := 7351.122, [191].log_data[50].time := 3600.0, [191].log_data[50].minminute := 56, [191].log_data[50].valid := 1, [191].log_data[51].time := 3600.0, [191].log_data[51].valid := 1, [191].log_data[52].min := -2.9400024, [191].log_data[52].max := 0.13999939, [191].log_data[52].total := -7346.108, [191].log_data[52].time := 3600.0, [191].log_data[52].minminute := 27,
        [191].log_data[52].maxminute := 5, [191].log_data[52].valid := 1, [191].log_data[53].min := -2.4800034, [191].log_data[53].max := 0.22000122, [191].log_data[53].total := -6860.3633, [191].log_data[53].time := 3600.0, [191].log_data[53].minminute := 2, [191].log_data[53].maxminute := 40, [191].log_data[53].valid := 1, [191].log_data[54].max := 0.543, [191].log_data[54].total := 1178.8529, [191].log_data[54].time := 3600.0, [191].log_data[54].minminute := 5, [191].log_data[54].maxminute := 27, [191].log_data[54].valid := 1, [191].log_data[55].max := 0.49800003, [191].log_data[55].total := 1178.3279, [191].log_data[55].time := 3600.0, [191].log_data[55].minminute := 7, [191].log_data[55].maxminute := 30, [191].log_data[55].valid := 1, [191].log_data[56].min := 0.16028486, [191].log_data[56].max := 0.16067745, [191].log_data[56].total := 577.6766, [191].log_data[56].time := 3600.0, [191].log_data[56].minminute := 34, [191].log_data[56].maxminute := 7, [191].log_data[56].valid := 1, [191].log_data[57].min := 0.3318828, [191].log_data[57].max := 0.3322754, [191].log_data[57].total := 1195.2809, [191].log_data[57].time := 3600.0, [191].log_data[57].minminute := 10, [191].log_data[57].valid := 1, [191].log_data[58].time := 3600.0, [191].log_data[58].valid := 1, [191].log_data[59].time := 3600.0, [191].log_data[59].valid := 1, [191].log_data[60].valid := 1, [191].log_data[61].valid := 1, [191].log_data[62].valid := 1, [191].log_data[63].valid := 1, [191].log_data[64].valid := 1, [191].log_data[65].valid := 1, [191].log_data[66].valid := 1, [191].log_data[67].valid := 1, [191].log_data[68].valid := 1, [191].log_data[69].valid := 1, [191].log_data[70].valid := 1, [191].log_data[71].valid := 1, [191].log_data[72].valid := 1, [191].log_data[73].valid := 1, [191].log_data[74].valid := 1, [191].log_data[75].valid := 1, [191].log_data[76].valid := 1, [191].log_data[77].valid := 1, [191].log_data[78].valid := 1, [191].log_data[79].valid := 1, [191].log_data[80].valid := 1, [191].log_data[81].valid := 1,
        [191].log_data[82].valid := 1, [191].log_data[83].valid := 1, [191].log_data[84].valid := 1, [191].log_data[85].valid := 1, [191].log_data[86].valid := 1, [191].log_data[87].valid := 1, [191].log_data[88].valid := 1, [191].log_data[89].valid := 1, [191].log_data[90].valid := 1, [191].log_data[91].valid := 1, [191].log_data[92].valid := 1, [191].log_data[93].valid := 1, [191].log_data[94].valid := 1, [191].log_data[95].valid := 1, [191].log_data[96].valid := 1, [191].log_data[97].valid := 1, [191].log_data[98].valid := 1, [191].log_data[99].valid := 1, [191].log_data[100].valid := 1, [191].log_data[101].valid := 1, [191].log_data[102].valid := 1, [191].log_data[103].valid := 1, [191].log_data[104].valid := 1, [191].log_data[105].valid := 1, [191].log_data[106].valid := 1, [191].log_data[107].valid := 1, [191].log_data[108].valid := 1, [191].log_data[109].valid := 1, [191].log_data[110].valid := 1, [191].log_data[111].valid := 1, [191].log_data[112].valid := 1, [191].log_data[113].valid := 1, [191].log_data[114].valid := 1, [191].log_data[115].valid := 1, [191].log_data[116].valid := 1, [191].log_data[117].valid := 1, [191].log_data[118].valid := 1, [191].log_data[119].valid := 1, [191].log_data[120].valid := 1, [191].log_data[121].valid := 1, [191].log_data[122].valid := 1, [191].log_data[123].valid := 1, [191].log_data[124].valid := 1, [191].time.Year := 2023, [191].time.Month := 1, [191].time.Day := 12, [191].time.Hour := 18, [191].time.Minute := 59, [191].time.Second := 59, [192].log_data[0].min := 1.0, [192].log_data[0].max := 1.0, [192].log_data[0].total := 3600.0, [192].log_data[0].time := 3600.0, [192].log_data[0].valid := 1, [192].log_data[1].max := 1.0, [192].log_data[1].total := 459.251, [192].log_data[1].time := 3600.0, [192].log_data[1].minminute := 7, [192].log_data[1].valid := 1, [192].log_data[2].max := 1.0,
